C02439=-605,59585,-14,-1321,-34531,-989
C02440=-605,59585,1386,-1321,-34531,-989
C02441=-133,59559,1353,-1384,-34516,-1179
C02442=-133,59559,-47,-1384,-34516,-1179
C02443=-94,59556,-50,-1389,-34515,-1194
C02444=-94,59556,1350,-1389,-34515,-1194
C02445=167,59542,1332,-1423,-34507,-1299
C02446=167,59542,-68,-1423,-34507,-1299
C02447=216,59539,-71,-1430,-34505,-1318
C02448=216,59539,1329,-1430,-34505,-1318
C02449=494,59523,1310,-1467,-34497,-1430
C02450=494,59523,-90,-1467,-34497,-1430
C02451=533,59521,-93,-1472,-34495,-1445
C02452=533,59521,1307,-1472,-34495,-1445
C02453=638,59515,1300,-1486,-34492,-1488
C02454=638,59515,-100,-1486,-34492,-1488
C02455=681,59512,-103,-1492,-34491,-1505
C02456=681,59512,1297,-1492,-34491,-1505
C02457=1167,59485,1263,-1556,-34476,-1699
C02458=1167,59485,-137,-1556,-34476,-1699
C02459=1205,59483,-140,-1561,-34474,-1715
C02460=1205,59483,1260,-1561,-34474,-1715
C02461=-5420,59813,1651,-682,-34655,941
C02462=-5420,59813,251,-682,-34655,941
C02463=-5370,59811,248,-689,-34654,922
C02464=-5370,59811,1648,-689,-34654,922
C02465=-4567,59765,1592,-795,-34629,600
C02466=-4567,59765,192,-795,-34629,600
C02467=-4511,59762,188,-803,-34627,577
C02468=-4511,59762,1588,-803,-34627,577
C02469=-4166,59743,1565,-849,-34616,439
C02470=-4166,59743,165,-849,-34616,439
C02471=-4106,59739,160,-857,-34614,415
C02472=-4106,59739,1560,-857,-34614,415
C02473=-3314,59694,1506,-962,-34589,97
C02474=-3314,59694,106,-962,-34589,97
C02475=-3268,59692,102,-968,-34588,79
C02476=-3268,59692,1502,-968,-34588,79
C02477=-2546,59651,1453,-1064,-34565,-211
C02478=-2546,59651,53,-1064,-34565,-211
C02479=-2500,59648,49,-1070,-34564,-229
C02480=-2500,59648,1449,-1070,-34564,-229
C02481=-2225,59633,1430,-1106,-34555,-339
C02482=-2225,59633,30,-1106,-34555,-339
C02483=-2173,59630,27,-1114,-34553,-360
C02484=-2173,59630,1427,-1114,-34553,-360
C02485=-1937,59617,1411,-1145,-34546,-455
C02486=-1937,59617,11,-1145,-34546,-455
C02487=-1891,59614,7,-1151,-34544,-473
C02488=-1891,59614,1407,-1151,-34544,-473
C02489=-1729,59605,1396,-1172,-34539,-538
C02490=-1729,59605,-4,-1172,-34539,-538
C02491=-1687,59602,-7,-1178,-34538,-555
C02492=-1687,59602,1393,-1178,-34538,-555
C02493=-1606,59598,1388,-1189,-34535,-588
C02494=-1606,59598,-12,-1189,-34535,-588
C02495=-1556,59595,-16,-1195,-34534,-607
C02496=-1556,59595,1384,-1195,-34534,-607
C02497=-1412,59587,1374,-1215,-34529,-665
C02498=-1412,59587,-26,-1215,-34529,-665
C02499=-1331,59582,-31,-1225,-34527,-698
C02500=-1331,59582,1369,-1225,-34527,-698
C02501=-1250,59578,1363,-1236,-34524,-730
C02502=-1250,59578,-37,-1236,-34524,-730
C02503=-1165,59573,-43,-1247,-34522,-764
C02504=-1165,59573,1357,-1247,-34522,-764
C02505=-1056,59567,1350,-1262,-34518,-808
C02506=-1056,59567,-50,-1262,-34518,-808
C02507=-1010,59564,-53,-1268,-34517,-826
C02508=-1010,59564,1347,-1268,-34517,-826
C02509=-655,59544,1322,-1315,-34506,-969
C02510=-655,59544,-78,-1315,-34506,-969
C02511=-619,59542,-80,-1320,-34504,-983
C02512=-619,59542,1320,-1320,-34504,-983
C02513=-130,59514,1286,-1385,-34489,-1179
C02514=-130,59514,-114,-1385,-34489,-1179
C02515=-95,59512,-117,-1390,-34488,-1193
C02516=-95,59512,1283,-1390,-34488,-1193
C02517=173,59497,1265,-1425,-34480,-1301
C02518=173,59497,-135,-1425,-34480,-1301
C02519=219,59495,-138,-1431,-34478,-1319
C02520=219,59495,1262,-1431,-34478,-1319
C02521=497,59479,1242,-1468,-34469,-1430
C02522=497,59479,-158,-1468,-34469,-1430
C02523=539,59477,-161,-1474,-34468,-1447
C02524=539,59477,1239,-1474,-34468,-1447
C02525=648,59470,1232,-1488,-34465,-1491
C02526=648,59470,-168,-1488,-34465,-1491
C02527=691,59468,-171,-1494,-34463,-1508
C02528=691,59468,1229,-1494,-34463,-1508
C02529=1170,59441,1196,-1557,-34448,-1700
C02530=1170,59441,-204,-1557,-34448,-1700
C02531=1208,59439,-207,-1563,-34447,-1716
C02532=1208,59439,1193,-1563,-34447,-1716
C02533=-5403,59768,1583,-685,-34628,935
C02534=-5403,59768,183,-685,-34628,935
C02535=-5354,59765,179,-692,-34626,915
C02536=-5354,59765,1579,-692,-34626,915
C02537=-4551,59720,1524,-798,-34601,594
C02538=-4551,59720,124,-798,-34601,594
C02539=-4494,59717,120,-806,-34599,571
C02540=-4494,59717,1520,-806,-34599,571
C02541=-4195,59700,1499,-846,-34590,451
C02542=-4195,59700,99,-846,-34590,451
C02543=-4128,59696,95,-854,-34588,424
C02544=-4128,59696,1495,-854,-34588,424
C02545=-3332,59651,1440,-960,-34563,105
C02546=-3332,59651,40,-960,-34563,105
C02547=-3283,59648,36,-967,-34561,85
C02548=-3283,59648,1436,-967,-34561,85
C02549=-2543,59607,1385,-1065,-34538,-211
C02550=-2543,59607,-15,-1065,-34538,-211
C02551=-2494,59604,-18,-1072,-34536,-231
C02552=-2494,59604,1382,-1072,-34536,-231
C02553=-2226,59589,1363,-1107,-34528,-338
C02554=-2226,59589,-37,-1107,-34528,-338
C02555=-2177,59586,-40,-1114,-34526,-358
C02556=-2177,59586,1360,-1114,-34526,-358
C02557=-1920,59571,1342,-1148,-34518,-461
C02558=-1920,59571,-58,-1148,-34518,-461
C02559=-1870,59569,-61,-1154,-34517,-481
C02560=-1870,59569,1339,-1154,-34517,-481
C02561=-1758,59562,1331,-1169,-34513,-526
C02562=-1758,59562,-69,-1169,-34513,-526
C02563=-1715,59560,-72,-1175,-34512,-543
C02564=-1715,59560,1328,-1175,-34512,-543
C02565=-1599,59553,1320,-1190,-34508,-590
C02566=-1599,59553,-80,-1190,-34508,-590
C02567=-1532,59549,-84,-1199,-34506,-616
C02568=-1532,59549,1316,-1199,-34506,-616
C02569=-1370,59540,1304,-1221,-34501,-681
C02570=-1370,59540,-96,-1221,-34501,-681
C02571=-1226,59532,-106,-1240,-34496,-739
C02572=-1226,59532,1294,-1240,-34496,-739
C02573=-1039,59522,1282,-1265,-34491,-814
C02574=-1039,59522,-118,-1265,-34491,-814
C02575=-986,59519,-122,-1272,-34489,-835
C02576=-986,59519,1278,-1272,-34489,-835
C02577=-684,59502,1257,-1312,-34479,-957
C02578=-684,59502,-143,-1312,-34479,-957
C02579=-641,59499,-146,-1318,-34478,-973
C02580=-641,59499,1254,-1318,-34478,-973
C02581=-131,59470,1219,-1386,-34462,-1178
C02582=-131,59470,-181,-1386,-34462,-1178
C02583=-92,59468,-184,-1391,-34461,-1194
C02584=-92,59468,1216,-1391,-34461,-1194
C02585=176,59453,1198,-1426,-34452,-1301
C02586=176,59453,-202,-1426,-34452,-1301
C02587=222,59450,-206,-1432,-34451,-1319
C02588=222,59450,1194,-1432,-34451,-1319
C02589=503,59435,1175,-1470,-34442,-1432
C02590=503,59435,-225,-1470,-34442,-1432
C02591=542,59432,-228,-1475,-34441,-1448
C02592=542,59432,1172,-1475,-34441,-1448
C02593=655,59426,1165,-1490,-34437,-1493
C02594=655,59426,-235,-1490,-34437,-1493
C02595=697,59424,-238,-1496,-34436,-1510
C02596=697,59424,1162,-1496,-34436,-1510
C02597=827,59416,1153,-1513,-34432,-1562
C02598=827,59416,-247,-1513,-34432,-1562
C02599=848,59415,-249,-1516,-34431,-1571
C02600=848,59415,1151,-1516,-34431,-1571
C02601=1165,59397,1129,-1558,-34421,-1698
C02602=1165,59397,-271,-1558,-34421,-1698
C02603=1204,59395,-273,-1563,-34420,-1713
C02604=1204,59395,1127,-1563,-34420,-1713
C02605=-5393,59723,1515,-687,-34601,932
C02606=-5393,59723,115,-687,-34601,932
C02607=-5341,59720,111,-694,-34599,911
C02608=-5341,59720,1511,-694,-34599,911
C02609=-4534,59675,1456,-801,-34574,587
C02610=-4534,59675,56,-801,-34574,587
C02611=-4474,59671,52,-809,-34572,563
C02612=-4474,59671,1452,-809,-34572,563
C02613=-4221,59657,1434,-843,-34564,462
C02614=-4221,59657,34,-843,-34564,462
C02615=-4157,59653,30,-851,-34562,436
C02616=-4157,59653,1430,-851,-34562,436
C02617=-3344,59607,1374,-959,-34536,110
C02618=-3344,59607,-26,-959,-34536,110
C02619=-3298,59605,-30,-965,-34535,92
C02620=-3298,59605,1370,-965,-34535,92
C02621=-2544,59562,1318,-1066,-34511,-210
C02622=-2544,59562,-82,-1066,-34511,-210
C02623=-2498,59560,-85,-1072,-34509,-229
C02624=-2498,59560,1315,-1072,-34509,-229
C02625=-2227,59544,1296,-1108,-34501,-337
C02626=-2227,59544,-104,-1108,-34501,-337
C02627=-2178,59542,-107,-1114,-34499,-357
C02628=-2178,59542,1293,-1114,-34499,-357
C02629=-1892,59526,1273,-1152,-34490,-471
C02630=-1892,59526,-127,-1152,-34490,-471
C02631=-1741,59517,-137,-1172,-34486,-532
C02632=-1741,59517,1263,-1172,-34486,-532
C02633=-1019,59476,1213,-1268,-34463,-822
C02634=-1019,59476,-187,-1268,-34463,-822
C02635=-941,59472,-192,-1279,-34460,-853
C02636=-941,59472,1208,-1279,-34460,-853
C02637=-723,59460,1193,-1308,-34453,-940
C02638=-723,59460,-207,-1308,-34453,-940
C02639=-667,59457,-211,-1315,-34452,-963
C02640=-667,59457,1189,-1315,-34452,-963
C02641=-135,59427,1152,-1386,-34435,-1176
C02642=-135,59427,-248,-1386,-34435,-1176
C02643=-89,59424,-251,-1392,-34433,-1194
C02644=-89,59424,1149,-1392,-34433,-1194
C02645=175,59409,1131,-1427,-34425,-1300
C02646=175,59409,-269,-1427,-34425,-1300
C02647=221,59406,-273,-1433,-34424,-1318
C02648=221,59406,1127,-1433,-34424,-1318
C02649=506,59390,1108,-1471,-34415,-1433
C02650=506,59390,-292,-1471,-34415,-1433
C02651=541,59388,-295,-1476,-34414,-1447
C02652=541,59388,1105,-1476,-34414,-1447
C02653=661,59382,1097,-1492,-34410,-1495
C02654=661,59382,-303,-1492,-34410,-1495
C02655=707,59379,-306,-1498,-34408,-1513
C02656=707,59379,1094,-1498,-34408,-1513
C02657=830,59372,1085,-1514,-34404,-1563
C02658=830,59372,-315,-1514,-34404,-1563
C02659=855,59371,-316,-1517,-34404,-1573
C02660=855,59371,1084,-1517,-34404,-1573
C02661=1154,59354,1063,-1557,-34394,-1693
C02662=1154,59354,-337,-1557,-34394,-1693
C02663=1197,59351,-340,-1563,-34393,-1710
C02664=1197,59351,1060,-1563,-34393,-1710
C02665=-5380,59678,1447,-689,-34573,927
C02666=-5380,59678,47,-689,-34573,927
C02667=-5320,59674,43,-697,-34571,903
C02668=-5320,59674,1443,-697,-34571,903
C02669=-4517,59629,1388,-804,-34546,581
C02670=-4517,59629,-12,-804,-34546,581
C02671=-4443,59625,-18,-814,-34544,552
C02672=-4443,59625,1382,-814,-34544,552
C02673=-4257,59614,1370,-839,-34538,477
C02674=-4257,59614,-30,-839,-34538,477
C02675=-4183,59610,-36,-849,-34536,447
C02676=-4183,59610,1364,-849,-34536,447
C02677=-3362,59564,1308,-958,-34510,118
C02678=-3362,59564,-92,-958,-34510,118
C02679=-3316,59562,-95,-964,-34508,100
C02680=-3316,59562,1305,-964,-34508,100
C02681=-2221,59500,1229,-1109,-34474,-339
C02682=-2221,59500,-171,-1109,-34474,-339
C02683=-2193,59498,-173,-1113,-34473,-351
C02684=-2193,59498,1227,-1113,-34473,-351
C02685=-991,59431,1144,-1273,-34435,-832
C02686=-991,59431,-256,-1273,-34435,-832
C02687=-699,59414,-276,-1312,-34426,-949
C02688=-699,59414,1124,-1312,-34426,-949
C02689=-136,59383,1085,-1386,-34408,-1175
C02690=-136,59383,-315,-1386,-34408,-1175
C02691=-86,59380,-318,-1393,-34406,-1195
C02692=-86,59380,1082,-1393,-34406,-1195
C02693=178,59365,1063,-1428,-34398,-1301
C02694=178,59365,-337,-1428,-34398,-1301
C02695=224,59362,-340,-1434,-34396,-1319
C02696=224,59362,1060,-1434,-34396,-1319
C02697=509,59346,1041,-1472,-34387,-1433
C02698=509,59346,-359,-1472,-34387,-1433
C02699=544,59344,-362,-1477,-34386,-1447
C02700=544,59344,1038,-1477,-34386,-1447
C02701=664,59337,1030,-1493,-34383,-1495
C02702=664,59337,-370,-1493,-34383,-1495
C02703=710,59335,-373,-1499,-34381,-1514
C02704=710,59335,1027,-1499,-34381,-1514
C02705=837,59328,1018,-1516,-34377,-1565
C02706=837,59328,-382,-1516,-34377,-1565
C02707=868,59326,-384,-1520,-34376,-1577
C02708=868,59326,1016,-1520,-34376,-1577
C02709=1136,59311,997,-1555,-34368,-1685
C02710=1136,59311,-403,-1555,-34368,-1685
C02711=1185,59308,-406,-1562,-34366,-1704
C02712=1185,59308,994,-1562,-34366,-1704
C02713=-5360,59632,1379,-693,-34546,920
C02714=-5360,59632,-21,-693,-34546,920
C02715=-5304,59629,-25,-700,-34544,897
C02716=-5304,59629,1375,-700,-34544,897
C02717=-4490,59583,1319,-808,-34518,571
C02718=-4490,59583,-81,-808,-34518,571
C02719=-4384,59577,-89,-822,-34515,529
C02720=-4384,59577,1311,-822,-34515,529
C02721=-4325,59574,1307,-830,-34513,505
C02722=-4325,59574,-93,-830,-34513,505
C02723=-4219,59568,-100,-844,-34510,462
C02724=-4219,59568,1300,-844,-34510,462
C02725=-3381,59521,1242,-956,-34483,126
C02726=-3381,59521,-158,-956,-34483,126
C02727=-3331,59518,-161,-962,-34482,106
C02728=-3331,59518,1239,-962,-34482,106
C02729=-901,59381,1071,-1285,-34405,-868
C02730=-901,59381,-329,-1285,-34405,-868
C02731=-784,59375,-337,-1301,-34401,-914
C02732=-784,59375,1063,-1301,-34401,-914
C02733=-126,59338,1017,-1389,-34380,-1178
C02734=-126,59338,-383,-1389,-34380,-1178
C02735=-94,59336,-385,-1393,-34379,-1191
C02736=-94,59336,1015,-1393,-34379,-1191
C02737=181,59321,996,-1429,-34371,-1301
C02738=181,59321,-404,-1429,-34371,-1301
C02739=227,59318,-407,-1435,-34369,-1320
C02740=227,59318,993,-1435,-34369,-1320
C02741=508,59302,974,-1473,-34360,-1432
C02742=508,59302,-426,-1473,-34360,-1432
C02743=561,59299,-430,-1480,-34359,-1454
C02744=561,59299,970,-1480,-34359,-1454
C02745=843,59283,951,-1517,-34350,-1567
C02746=843,59283,-449,-1517,-34350,-1567
C02747=878,59281,-452,-1522,-34349,-1581
C02748=878,59281,948,-1522,-34349,-1581
C02749=1107,59269,932,-1552,-34341,-1672
C02750=1107,59269,-468,-1552,-34341,-1672
C02751=1164,59265,-472,-1560,-34340,-1695
C02752=1164,59265,928,-1560,-34340,-1695
C02753=-5340,59586,1310,-696,-34518,912
C02754=-5340,59586,-90,-696,-34518,912
C02755=-5277,59583,-94,-704,-34516,887
C02756=-5277,59583,1306,-704,-34516,887
C02757=-4452,59537,1249,-814,-34490,556
C02758=-4452,59537,-151,-814,-34490,556
C02759=-4269,59526,-164,-838,-34484,483
C02760=-4269,59526,1236,-838,-34484,483
C02761=-3403,59478,1176,-954,-34457,136
C02762=-3403,59478,-224,-954,-34457,136
C02763=-3353,59475,-227,-960,-34455,116
C02764=-3353,59475,1173,-960,-34455,116
C02765=511,59258,906,-1474,-34333,-1433
C02766=511,59258,-494,-1474,-34333,-1433
C02767=561,59255,-497,-1481,-34331,-1453
C02768=561,59255,903,-1481,-34331,-1453
C02769=853,59239,883,-1519,-34322,-1570
C02770=853,59239,-517,-1519,-34322,-1570
C02771=902,59236,-521,-1526,-34321,-1590
C02772=902,59236,879,-1526,-34321,-1590
C02773=1057,59227,869,-1547,-34316,-1652
C02774=1057,59227,-531,-1547,-34316,-1652
C02775=1138,59223,-537,-1557,-34313,-1684
C02776=1138,59223,863,-1557,-34313,-1684
C02777=-5313,59540,1241,-700,-34490,902
C02778=-5313,59540,-159,-700,-34490,902
C02779=-5253,59537,-163,-708,-34489,878
C02780=-5253,59537,1237,-708,-34489,878
C02781=-3418,59434,1110,-952,-34430,142
C02782=-3418,59434,-290,-952,-34430,142
C02783=-3375,59432,-292,-958,-34429,125
C02784=-3375,59432,1108,-958,-34429,125
C02785=874,59194,814,-1523,-34294,-1578
C02786=874,59194,-586,-1523,-34294,-1578
C02787=1103,59181,-601,-1553,-34287,-1669
C02788=1103,59181,799,-1553,-34287,-1669
C02789=1508,59158,771,-1607,-34274,-1832
C02790=1508,59158,-629,-1607,-34274,-1832
C02791=1532,59157,-631,-1611,-34273,-1842
C02792=1532,59157,769,-1611,-34273,-1842
C02793=-5293,59495,1173,-704,-34463,894
C02794=-5293,59495,-227,-704,-34463,894
C02795=-5229,59491,-232,-712,-34461,869
C02796=-5229,59491,1168,-712,-34461,869
C02797=-3440,59391,1045,-950,-34404,151
C02798=-3440,59391,-355,-950,-34404,151
C02799=-3387,59388,-359,-957,-34402,130
C02800=-3387,59388,1041,-957,-34402,130
C02801=915,59148,745,-1529,-34266,-1594
C02802=915,59148,-655,-1529,-34266,-1594
C02803=1038,59141,-664,-1546,-34262,-1643
C02804=1038,59141,736,-1546,-34262,-1643
C02805=1482,59116,705,-1605,-34248,-1821
C02806=1482,59116,-695,-1605,-34248,-1821
C02807=1567,59111,-700,-1616,-34245,-1855
C02808=1567,59111,700,-1616,-34245,-1855
C02809=-5266,59449,1104,-708,-34435,884
C02810=-5266,59449,-296,-708,-34435,884
C02811=-5202,59445,-301,-716,-34433,858
C02812=-5202,59445,1099,-716,-34433,858
C02813=-3458,59348,979,-948,-34378,159
C02814=-3458,59348,-421,-948,-34378,159
C02815=-3405,59345,-424,-955,-34376,138
C02816=-3405,59345,976,-955,-34376,138
C02817=1485,59072,638,-1606,-34221,-1821
C02818=1485,59072,-762,-1606,-34221,-1821
C02819=1538,59069,-765,-1613,-34219,-1843
C02820=1538,59069,635,-1613,-34219,-1843
C02821=-5245,59403,1035,-711,-34408,876
C02822=-5245,59403,-365,-711,-34408,876
C02823=-5178,59399,-369,-720,-34405,849
C02824=-5178,59399,1031,-720,-34405,849
C02825=-3484,59305,914,-946,-34351,170
C02826=-3484,59305,-486,-946,-34351,170
C02827=-3424,59302,-490,-954,-34350,146
C02828=-3424,59302,910,-954,-34350,146
C02829=-5215,59357,966,-716,-34380,864
C02830=-5215,59357,-434,-716,-34380,864
C02831=-5155,59354,-438,-724,-34378,840
C02832=-5155,59354,962,-724,-34378,840
C02833=-3516,59262,849,-942,-34325,184
C02834=-3516,59262,-551,-942,-34325,184
C02835=-3460,59259,-555,-949,-34324,161
C02836=-3460,59259,845,-949,-34324,161
C02837=-5184,59311,897,-721,-34352,853
C02838=-5184,59311,-503,-721,-34352,853
C02839=-5117,59307,-508,-730,-34350,826
C02840=-5117,59307,892,-730,-34350,826
C02841=-3552,59220,784,-938,-34300,199
C02842=-3552,59220,-616,-938,-34300,199
C02843=-3482,59216,-620,-947,-34297,171
C02844=-3482,59216,780,-947,-34297,171
C02845=-5157,59265,828,-725,-34324,842
C02846=-5157,59265,-572,-725,-34324,842
C02847=-5076,59260,-578,-736,-34321,810
C02848=-5076,59260,822,-736,-34321,810
C02849=-3592,59178,720,-933,-34274,215
C02850=-3592,59178,-680,-933,-34274,215
C02851=-3518,59174,-685,-943,-34272,186
C02852=-3518,59174,715,-943,-34272,186
C02853=-5119,59218,758,-731,-34296,828
C02854=-5119,59218,-642,-731,-34296,828
C02855=-5041,59214,-647,-741,-34293,797
C02856=-5041,59214,753,-741,-34293,797
C02857=-3635,59136,656,-928,-34248,233
C02858=-3635,59136,-744,-928,-34248,233
C02859=-3558,59132,-749,-939,-34246,202
C02860=-3558,59132,651,-939,-34246,202
C02861=-5081,59172,689,-736,-34268,813
C02862=-5081,59172,-711,-736,-34268,813
C02863=-4965,59165,-719,-752,-34264,766
C02864=-4965,59165,681,-752,-34264,766
C02865=-3678,59094,592,-923,-34223,251
C02866=-3678,59094,-808,-923,-34223,251
C02867=-3597,59090,-814,-934,-34220,219
C02868=-3597,59090,586,-934,-34220,219
C02869=-5036,59125,618,-743,-34239,796
C02870=-5036,59125,-782,-743,-34239,796
C02871=-4888,59117,-792,-763,-34234,736
C02872=-4888,59117,608,-763,-34234,736
C02873=-3736,59053,529,-916,-34197,275
C02874=-3736,59053,-871,-916,-34197,275
C02875=-3648,59048,-877,-928,-34195,239
C02876=-3648,59048,523,-928,-34195,239
C02877=-4953,59076,546,-755,-34210,763
C02878=-4953,59076,-854,-755,-34210,763
C02879=-4819,59068,-864,-773,-34205,709
C02880=-4819,59068,536,-773,-34205,709
C02881=-3782,59011,465,-911,-34172,294
C02882=-3782,59011,-935,-911,-34172,294
C02883=-3694,59006,-941,-922,-34169,259
C02884=-3694,59006,459,-922,-34169,259
C02885=-4880,59027,473,-765,-34180,734
C02886=-4880,59027,-927,-765,-34180,734
C02887=-4739,59019,-936,-784,-34176,677
C02888=-4739,59019,464,-784,-34176,677
C02889=-3840,58970,402,-904,-34147,317
C02890=-3840,58970,-998,-904,-34147,317
C02891=-3748,58965,-1004,-916,-34144,281
C02892=-3748,58965,396,-916,-34144,281
C02893=-4800,58978,401,-777,-34151,702
C02894=-4800,58978,-999,-777,-34151,702
C02895=-4609,58968,-1012,-802,-34145,626
C02896=-4609,58968,388,-802,-34145,626
C02897=-3925,58930,341,-893,-34123,352
C02898=-3925,58930,-1059,-893,-34123,352
C02899=-3802,58923,-1068,-910,-34119,303
C02900=-3802,58923,332,-910,-34119,303
C02901=-4695,58928,327,-791,-34120,661
C02902=-4695,58928,-1073,-791,-34120,661
C02903=-4462,58915,-1089,-822,-34113,568
C02904=-4462,58915,311,-822,-34113,568
C02905=-4194,58901,292,-858,-34104,460
C02906=-4194,58901,-1108,-858,-34104,460
C02907=-3873,58883,-1130,-901,-34094,332
C02908=-3873,58883,270,-901,-34094,332
C02909=-4537,58875,249,-813,-34088,598
C02910=-4537,58875,-1151,-813,-34088,598
C02911=-3991,58845,-1189,-886,-34071,379
C02912=-3991,58845,211,-886,-34071,379
C02913=-4485,58828,178,-821,-34060,578
C02914=-4485,58828,-1222,-821,-34060,578
C02915=-4330,58819,-1233,-841,-34055,516
C02916=-4330,58819,167,-841,-34055,516
C02917=-4493,58784,112,-820,-34033,582
C02918=-4493,58784,-1288,-820,-34033,582
C02919=-4430,58780,-1293,-829,-34031,556
C02920=-4430,58780,107,-829,-34031,556
C02921=-4494,58739,44,-821,-34006,583
C02922=-4494,58739,-1356,-821,-34006,583
C02923=-4427,58736,-1360,-830,-34004,556
C02924=-4427,58736,40,-830,-34004,556
C02925=-4492,58695,-23,-822,-33979,582
C02926=-4492,58695,-1423,-822,-33979,582
C02927=-4428,58691,-1427,-830,-33977,557
C02928=-4428,58691,-27,-830,-33977,557
C02929=-4478,58650,-91,-824,-33952,577
C02930=-4478,58650,-1491,-824,-33952,577
C02931=-4422,58647,-1495,-832,-33950,555
C02932=-4422,58647,-95,-832,-33950,555
C02933=-4472,58605,-158,-826,-33924,576
C02934=-4472,58605,-1558,-826,-33924,576
C02935=-4388,58600,-1564,-837,-33922,542
C02936=-4388,58600,-164,-837,-33922,542
C02937=-4473,58560,-225,-826,-33898,576
C02938=-4473,58560,-1625,-826,-33898,576
C02939=-4371,58555,-1632,-840,-33894,535
C02940=-4371,58555,-232,-840,-33894,535
C02941=-4485,58517,-292,-825,-33871,582
C02942=-4485,58517,-1692,-825,-33871,582
C02943=-4344,58509,-1701,-844,-33866,525
C02944=-4344,58509,-301,-844,-33866,525
C02945=-4503,58473,-357,-824,-33845,590
C02946=-4503,58473,-1757,-824,-33845,590
C02947=-4419,58469,-1763,-835,-33842,556
C02948=-4419,58469,-363,-835,-33842,556
C02949=-4387,58467,-365,-839,-33841,543
C02950=-4387,58467,-1765,-839,-33841,543
C02951=-4309,58463,-1771,-849,-33838,512
C02952=-4309,58463,-371,-849,-33838,512
C02953=-4526,58430,-423,-821,-33818,599
C02954=-4526,58430,-1823,-821,-33818,599
C02955=-4416,58424,-1830,-836,-33815,555
C02956=-4416,58424,-430,-836,-33815,555
C02957=-4349,58421,-435,-845,-33813,528
C02958=-4349,58421,-1835,-845,-33813,528
C02959=-4279,58417,-1840,-854,-33810,500
C02960=-4279,58417,-440,-854,-33810,500
C02961=-4548,58387,-488,-819,-33792,608
C02962=-4548,58387,-1888,-819,-33792,608
C02963=-4491,58384,-1892,-827,-33790,586
C02964=-4491,58384,-492,-827,-33790,586
C02965=-4463,58382,-494,-830,-33789,574
C02966=-4463,58382,-1894,-830,-33789,574
C02967=-4417,58380,-1897,-836,-33788,556
C02968=-4417,58380,-497,-836,-33788,556
C02969=-4315,58374,-504,-850,-33785,515
C02970=-4315,58374,-1904,-850,-33785,515
C02971=-4244,58370,-1909,-859,-33782,487
C02972=-4244,58370,-509,-859,-33782,487
C02973=-4570,58344,-554,-817,-33766,618
C02974=-4570,58344,-1954,-817,-33766,618
C02975=-4510,58340,-1958,-825,-33764,594
C02976=-4510,58340,-558,-825,-33764,594
C02977=-4464,58338,-561,-831,-33762,575
C02978=-4464,58338,-1961,-831,-33762,575
C02979=-4418,58335,-1964,-837,-33761,557
C02980=-4418,58335,-564,-837,-33761,557
C02981=-4284,58328,-574,-855,-33757,503
C02982=-4284,58328,-1974,-855,-33757,503
C02983=-4213,58324,-1978,-864,-33754,475
C02984=-4213,58324,-578,-864,-33754,475
C02985=-4599,58301,-619,-813,-33740,630
C02986=-4599,58301,-2019,-813,-33740,630
C02987=-4546,58298,-2023,-821,-33738,609
C02988=-4546,58298,-623,-821,-33738,609
C02989=-4461,58293,-628,-832,-33735,575
C02990=-4461,58293,-2028,-832,-33735,575
C02991=-4415,58291,-2032,-838,-33734,557
C02992=-4415,58291,-632,-838,-33734,557
C02993=-4250,58282,-643,-860,-33728,490
C02994=-4250,58282,-2043,-860,-33728,490
C02995=-4186,58279,-2047,-869,-33726,465
C02996=-4186,58279,-647,-869,-33726,465
C02997=-4621,58257,-685,-811,-33714,639
C02998=-4621,58257,-2085,-811,-33714,639
C02999=-4575,58255,-2088,-817,-33712,621
C03000=-4575,58255,-688,-817,-33712,621
C03001=-4459,58249,-696,-833,-33708,574
C03002=-4459,58249,-2096,-833,-33708,574
C03003=-4416,58246,-2099,-839,-33707,557
C03004=-4416,58246,-699,-839,-33707,557
C03005=-4222,58236,-712,-864,-33701,480
C03006=-4222,58236,-2112,-864,-33701,480
C03007=-4152,58232,-2117,-874,-33698,452
C03008=-4152,58232,-717,-874,-33698,452
C03009=-4650,58215,-750,-808,-33688,652
C03010=-4650,58215,-2150,-808,-33688,652
C03011=-4597,58212,-2153,-815,-33686,630
C03012=-4597,58212,-753,-815,-33686,630
C03013=-4460,58204,-763,-833,-33681,575
C03014=-4460,58204,-2163,-833,-33681,575
C03015=-4421,58202,-2165,-839,-33680,560
C03016=-4421,58202,-765,-839,-33680,560
C03017=-4188,58190,-781,-870,-33672,467
C03018=-4188,58190,-2181,-870,-33672,467
C03019=-4107,58185,-2187,-881,-33670,434
C03020=-4107,58185,-787,-881,-33670,434
C03021=-4683,58172,-815,-804,-33662,665
C03022=-4683,58172,-2215,-804,-33662,665
C03023=-4627,58169,-2218,-812,-33660,643
C03024=-4627,58169,-818,-812,-33660,643
C03025=-4461,58160,-830,-834,-33654,576
C03026=-4461,58160,-2230,-834,-33654,576
C03027=-4418,58158,-2233,-840,-33653,559
C03028=-4418,58158,-833,-840,-33653,559
C03029=-4150,58143,-851,-875,-33644,452
C03030=-4150,58143,-2251,-875,-33644,452
C03031=-4069,58139,-2257,-886,-33642,419
C03032=-4069,58139,-857,-886,-33642,419
C03033=-4716,58129,-879,-801,-33636,679
C03034=-4716,58129,-2279,-801,-33636,679
C03035=-4659,58126,-2283,-808,-33634,656
C03036=-4659,58126,-883,-808,-33634,656
C03037=-4458,58115,-897,-835,-33627,576
C03038=-4458,58115,-2297,-835,-33627,576
C03039=-4419,58113,-2300,-840,-33626,560
C03040=-4419,58113,-900,-840,-33626,560
C03041=-4102,58096,-921,-883,-33616,433
C03042=-4102,58096,-2321,-883,-33616,433
C03043=-4035,58093,-2326,-892,-33613,406
C03044=-4035,58093,-926,-892,-33613,406
C03045=-4745,58086,-944,-797,-33610,691
C03046=-4745,58086,-2344,-797,-33610,691
C03047=-4692,58084,-2348,-804,-33608,670
C03048=-4692,58084,-948,-804,-33608,670
C03049=-4459,58071,-964,-836,-33600,577
C03050=-4459,58071,-2364,-836,-33600,577
C03051=-4417,58069,-2367,-841,-33599,560
C03052=-4417,58069,-967,-841,-33599,560
C03053=-4064,58050,-991,-888,-33587,418
C03054=-4064,58050,-2391,-888,-33587,418
C03055=-3990,58046,-2396,-898,-33585,389
C03056=-3990,58046,-996,-898,-33585,389
C03057=-4785,58044,-1009,-793,-33584,708
C03058=-4785,58044,-2409,-793,-33584,708
C03059=-4725,58041,-2413,-801,-33582,683
C03060=-4725,58041,-1013,-801,-33582,683
C03061=-4456,58027,-1031,-837,-33573,576
C03062=-4456,58027,-2431,-837,-33573,576
C03063=-4414,58024,-2434,-842,-33572,559
C03064=-4414,58024,-1034,-842,-33572,559
C03065=-4019,58003,-1061,-895,-33559,401
C03066=-4019,58003,-2461,-895,-33559,401
C03067=-3938,57999,-2467,-906,-33556,369
C03068=-3938,57999,-1067,-906,-33556,369
C03069=-4817,58001,-1074,-789,-33558,721
C03070=-4817,58001,-2474,-789,-33558,721
C03071=-4765,57998,-2477,-796,-33557,700
C03072=-4765,57998,-1077,-796,-33557,700
C03073=-4454,57982,-1099,-838,-33546,576
C03074=-4454,57982,-2499,-838,-33546,576
C03075=-4411,57980,-2501,-843,-33545,559
C03076=-4411,57980,-1101,-843,-33545,559
C03077=-3977,57957,-1131,-901,-33531,385
C03078=-3977,57957,-2531,-901,-33531,385
C03079=-3900,57953,-2536,-912,-33528,354
C03080=-3900,57953,-1136,-912,-33528,354
C03081=-4850,57959,-1138,-785,-33533,735
C03082=-4850,57959,-2538,-785,-33533,735
C03083=-4797,57956,-2542,-792,-33531,714
C03084=-4797,57956,-1142,-792,-33531,714
C03085=-4455,57938,-1166,-838,-33519,577
C03086=-4455,57938,-2566,-838,-33519,577
C03087=-4412,57935,-2568,-844,-33518,560
C03088=-4412,57935,-1168,-844,-33518,560
C03089=-3936,57910,-1201,-908,-33502,369
C03090=-3936,57910,-2601,-908,-33502,369
C03091=-3858,57906,-2606,-918,-33500,338
C03092=-3858,57906,-1206,-918,-33500,338
C03093=-4887,57916,-1203,-781,-33507,750
C03094=-4887,57916,-2603,-781,-33507,750
C03095=-4837,57913,-2606,-788,-33505,730
C03096=-4837,57913,-1206,-788,-33505,730
C03097=-4452,57893,-1233,-839,-33492,576
C03098=-4452,57893,-2633,-839,-33492,576
C03099=-4413,57891,-2635,-844,-33491,561
C03100=-4413,57891,-1235,-844,-33491,561
C03101=-3894,57864,-1271,-914,-33474,353
C03102=-3894,57864,-2671,-914,-33474,353
C03103=-3817,57859,-2676,-924,-33471,322
C03104=-3817,57859,-1276,-924,-33471,322
C03105=-4923,57874,-1268,-777,-33481,765
C03106=-4923,57874,-2668,-777,-33481,765
C03107=-4870,57871,-2671,-784,-33479,744
C03108=-4870,57871,-1271,-784,-33479,744
C03109=-4453,57849,-1300,-840,-33465,577
C03110=-4453,57849,-2700,-840,-33465,577
C03111=-4414,57847,-2702,-845,-33464,561
C03112=-4414,57847,-1302,-845,-33464,561
C03113=-3856,57817,-1341,-920,-33446,338
C03114=-3856,57817,-2741,-920,-33446,338
C03115=-3765,57812,-2747,-932,-33443,302
C03116=-3765,57812,-1347,-932,-33443,302
C03117=-4963,57831,-1332,-772,-33455,781
C03118=-4963,57831,-2732,-772,-33455,781
C03119=-4906,57828,-2736,-780,-33454,759
C03120=-4906,57828,-1336,-780,-33454,759
C03121=-4451,57804,-1367,-841,-33438,576
C03122=-4451,57804,-2767,-841,-33438,576
C03123=-4412,57802,-2770,-846,-33437,561
C03124=-4412,57802,-1370,-846,-33437,561
C03125=-3819,57771,-1410,-925,-33417,324
C03126=-3819,57771,-2810,-925,-33417,324
C03127=-3730,57766,-2816,-937,-33414,288
C03128=-3730,57766,-1416,-937,-33414,288
C03129=-5006,57789,-1396,-767,-33430,799
C03130=-5006,57789,-2796,-767,-33430,799
C03131=-4946,57786,-2800,-775,-33428,775
C03132=-4946,57786,-1400,-775,-33428,775
C03133=-4452,57760,-1434,-841,-33411,577
C03134=-4452,57760,-2834,-841,-33411,577
C03135=-4413,57758,-2837,-847,-33410,562
C03136=-4413,57758,-1437,-847,-33410,562
C03137=-3784,57725,-1480,-931,-33389,310
C03138=-3784,57725,-2880,-931,-33389,310
C03139=-3692,57720,-2886,-943,-33386,274
C03140=-3692,57720,-1486,-943,-33386,274
C03141=-5049,57747,-1460,-762,-33404,817
C03142=-5049,57747,-2860,-762,-33404,817
C03143=-4989,57744,-2864,-770,-33402,793
C03144=-4989,57744,-1464,-770,-33402,793
C03145=-4449,57715,-1501,-842,-33384,577
C03146=-4449,57715,-2901,-842,-33384,577
C03147=-4407,57713,-2904,-848,-33383,560
C03148=-4407,57713,-1504,-848,-33383,560
C03149=-3746,57678,-1549,-936,-33361,296
C03150=-3746,57678,-2949,-936,-33361,296
C03151=-3654,57673,-2956,-949,-33358,259
C03152=-3654,57673,-1556,-949,-33358,259
C03153=-5089,57704,-1525,-757,-33379,834
C03154=-5089,57704,-2925,-757,-33379,834
C03155=-5033,57701,-2928,-765,-33377,811
C03156=-5033,57701,-1528,-765,-33377,811
C03157=-4446,57671,-1569,-843,-33357,576
C03158=-4446,57671,-2969,-843,-33357,576
C03159=-4404,57668,-2971,-849,-33356,559
C03160=-4404,57668,-1571,-849,-33356,559
C03161=-3708,57632,-1619,-942,-33333,281
C03162=-3708,57632,-3019,-942,-33333,281
C03163=-3623,57627,-3025,-953,-33330,247
C03164=-3623,57627,-1625,-953,-33330,247
C03165=-5125,57662,-1589,-753,-33353,849
C03166=-5125,57662,-2989,-753,-33353,849
C03167=-5069,57659,-2993,-761,-33351,826
C03168=-5069,57659,-1593,-761,-33351,826
C03169=-4447,57626,-1636,-844,-33330,577
C03170=-4447,57626,-3036,-844,-33330,577
C03171=-4405,57624,-3038,-850,-33329,560
C03172=-4405,57624,-1638,-850,-33329,560
C03173=-3674,57586,-1688,-947,-33304,268
C03174=-3674,57586,-3088,-947,-33304,268
C03175=-3578,57581,-3095,-960,-33301,230
C03176=-3578,57581,-1695,-960,-33301,230
C03177=-5165,57619,-1654,-748,-33328,865
C03178=-5165,57619,-3054,-748,-33328,865
C03179=-5105,57616,-3058,-757,-33326,841
C03180=-5105,57616,-1658,-757,-33326,841
C03181=-4445,57582,-1703,-845,-33303,577
C03182=-4445,57582,-3103,-845,-33303,577
C03183=-4402,57580,-3106,-851,-33302,560
C03184=-4402,57580,-1706,-851,-33302,560
C03185=-3650,57540,-1757,-951,-33277,259
C03186=-3650,57540,-3157,-951,-33277,259
C03187=-3590,57537,-3161,-959,-33275,235
C03188=-3590,57537,-1761,-959,-33275,235
C03189=-5202,57577,-1718,-744,-33302,880
C03190=-5202,57577,-3118,-744,-33302,880
C03191=-5138,57574,-3122,-753,-33300,855
C03192=-5138,57574,-1722,-753,-33300,855
C03193=-4442,57537,-1770,-846,-33276,576
C03194=-4442,57537,-3170,-846,-33276,576
C03195=-4407,57535,-3172,-851,-33275,562
C03196=-4407,57535,-1772,-851,-33275,562
C03197=-3676,57497,-1822,-949,-33251,270
C03198=-3676,57497,-3222,-949,-33251,270
C03199=-3608,57494,-3227,-958,-33248,243
C03200=-3608,57494,-1827,-958,-33248,243
C03201=-5231,57534,-1783,-741,-33276,892
C03202=-5231,57534,-3183,-741,-33276,892
C03203=-5178,57531,-3187,-748,-33274,871
C03204=-5178,57531,-1787,-748,-33274,871
C03205=-4443,57493,-1837,-847,-33249,577
C03206=-4443,57493,-3237,-847,-33249,577
C03207=-4401,57491,-3240,-852,-33248,560
C03208=-4401,57491,-1840,-852,-33248,560
C03209=-3701,57454,-1888,-946,-33224,281
C03210=-3701,57454,-3288,-946,-33224,281
C03211=-3631,57450,-3293,-955,-33222,252
C03212=-3631,57450,-1893,-955,-33222,252
C03213=-5264,57491,-1848,-737,-33250,906
C03214=-5264,57491,-3248,-737,-33250,906
C03215=-5211,57488,-3252,-744,-33248,885
C03216=-5211,57488,-1852,-744,-33248,885
C03217=-4444,57448,-1904,-847,-33222,578
C03218=-4444,57448,-3304,-847,-33222,578
C03219=-4402,57446,-3307,-853,-33221,561
C03220=-4402,57446,-1907,-853,-33221,561
C03221=-3734,57411,-1953,-942,-33198,294
C03222=-3734,57411,-3353,-942,-33198,294
C03223=-3660,57408,-3358,-952,-33196,265
C03224=-3660,57408,-1958,-952,-33196,265
C03225=-5300,57449,-1913,-733,-33224,921
C03226=-5300,57449,-3313,-733,-33224,921
C03227=-5240,57445,-3317,-741,-33222,897
C03228=-5240,57445,-1917,-741,-33222,897
C03229=-4441,57404,-1971,-848,-33195,578
C03230=-4441,57404,-3371,-848,-33195,578
C03231=-4399,57402,-3374,-854,-33194,561
C03232=-4399,57402,-1974,-854,-33194,561
C03233=-3763,57369,-2018,-939,-33172,306
C03234=-3763,57369,-3418,-939,-33172,306
C03235=-3696,57365,-3422,-948,-33170,280
C03236=-3696,57365,-2022,-948,-33170,280
C03237=-5333,57406,-1977,-729,-33198,935
C03238=-5333,57406,-3377,-729,-33198,935
C03239=-5269,57402,-3382,-738,-33196,909
C03240=-5269,57402,-1982,-738,-33196,909
C03241=-4439,57359,-2039,-849,-33168,577
C03242=-4439,57359,-3439,-849,-33168,577
C03243=-4396,57357,-3441,-855,-33167,560
C03244=-4396,57357,-2041,-855,-33167,560
C03245=-3803,57326,-2082,-934,-33147,323
C03246=-3803,57326,-3482,-934,-33147,323
C03247=-3736,57323,-3487,-943,-33145,296
C03248=-3736,57323,-2087,-943,-33145,296
C03249=-5366,57363,-2042,-726,-33173,948
C03250=-5366,57363,-3442,-726,-33173,948
C03251=-5302,57360,-3447,-734,-33171,923
C03252=-5302,57360,-2047,-734,-33171,923
C03253=-4440,57315,-2106,-850,-33141,578
C03254=-4440,57315,-3506,-850,-33141,578
C03255=-4397,57313,-3508,-855,-33140,561
C03256=-4397,57313,-2108,-855,-33140,561
C03257=-3836,57284,-2147,-931,-33121,337
C03258=-3836,57284,-3547,-931,-33121,337
C03259=-3776,57281,-3551,-939,-33119,313
C03260=-3776,57281,-2151,-939,-33119,313
C03261=-5381,57319,-2108,-724,-33146,955
C03262=-5381,57319,-3508,-724,-33146,955
C03263=-5275,57314,-3516,-738,-33143,912
C03264=-5275,57314,-2116,-738,-33143,912
C03265=-4441,57271,-2173,-850,-33114,579
C03266=-4441,57271,-3573,-850,-33114,579
C03267=-4398,57268,-3575,-856,-33113,562
C03268=-4398,57268,-2175,-856,-33113,562
C03269=-3872,57241,-2211,-926,-33095,352
C03270=-3872,57241,-3611,-926,-33095,352
C03271=-3812,57238,-3615,-935,-33093,328
C03272=-3812,57238,-2215,-935,-33093,328
C03273=-5346,57273,-2178,-730,-33118,942
C03274=-5346,57273,-3578,-730,-33118,942
C03275=-5233,57267,-3586,-745,-33114,896
C03276=-5233,57267,-2186,-745,-33114,896
C03277=-4438,57226,-2240,-851,-33087,579
C03278=-4438,57226,-3640,-851,-33087,579
C03279=-4396,57224,-3643,-857,-33086,562
C03280=-4396,57224,-2243,-857,-33086,562
C03281=-3905,57199,-2276,-923,-33069,365
C03282=-3905,57199,-3676,-923,-33069,365
C03283=-3852,57196,-3680,-930,-33067,344
C03284=-3852,57196,-2280,-930,-33067,344
C03285=-5284,57225,-2249,-739,-33089,917
C03286=-5284,57225,-3649,-739,-33089,917
C03287=-5181,57220,-3656,-752,-33086,876
C03288=-5181,57220,-2256,-752,-33086,876
C03289=-4439,57182,-2307,-852,-33060,579
C03290=-4439,57182,-3707,-852,-33060,579
C03291=-4397,57180,-3710,-857,-33059,562
C03292=-4397,57180,-2310,-857,-33059,562
C03293=-3948,57156,-2340,-918,-33044,383
C03294=-3948,57156,-3740,-918,-33044,383
C03295=-3884,57153,-3745,-926,-33042,358
C03296=-3884,57153,-2345,-926,-33042,358
C03297=-5228,57178,-2320,-747,-33060,895
C03298=-5228,57178,-3720,-747,-33060,895
C03299=-5126,57173,-3727,-760,-33057,854
C03300=-5126,57173,-2327,-760,-33057,854
C03301=-4437,57137,-2374,-853,-33033,579
C03302=-4437,57137,-3774,-853,-33033,579
C03303=-4398,57135,-3777,-858,-33032,563
C03304=-4398,57135,-2377,-858,-33032,563
C03305=-3991,57114,-2404,-913,-33018,401
C03306=-3991,57114,-3804,-913,-33018,401
C03307=-3928,57111,-3809,-921,-33016,376
C03308=-3928,57111,-2409,-921,-33016,376
C03309=-5169,57130,-2391,-755,-33031,872
C03310=-5169,57130,-3791,-755,-33031,872
C03311=-5067,57125,-3798,-769,-33028,831
C03312=-5067,57125,-2398,-769,-33028,831
C03313=-4434,57093,-2441,-854,-33006,578
C03314=-4434,57093,-3841,-854,-33006,578
C03315=-4399,57091,-3844,-859,-33005,564
C03316=-4399,57091,-2444,-859,-33005,564
C03317=-4038,57072,-2468,-907,-32993,420
C03318=-4038,57072,-3868,-907,-32993,420
C03319=-3971,57069,-3873,-916,-32991,393
C03320=-3971,57069,-2473,-916,-32991,393
C03321=-5114,57083,-2462,-763,-33002,851
C03322=-5114,57083,-3862,-763,-33002,851
C03323=-5000,57077,-3870,-779,-32999,805
C03324=-5000,57077,-2470,-779,-32999,805
C03325=-4435,57048,-2508,-854,-32979,579
C03326=-4435,57048,-3908,-854,-32979,579
C03327=-4396,57046,-3911,-860,-32978,564
C03328=-4396,57046,-2511,-860,-32978,564
C03329=-4081,57030,-2532,-902,-32967,438
C03330=-4081,57030,-3932,-902,-32967,438
C03331=-4021,57027,-3936,-910,-32965,414
C03332=-4021,57027,-2536,-910,-32965,414
C03333=-5058,57036,-2533,-772,-32974,829
C03334=-5058,57036,-3933,-772,-32974,829
C03335=-4938,57030,-3941,-788,-32970,781
C03336=-4938,57030,-2541,-788,-32970,781
C03337=-4436,57004,-2575,-855,-32952,580
C03338=-4436,57004,-3975,-855,-32952,580
C03339=-4397,57002,-3978,-860,-32951,565
C03340=-4397,57002,-2578,-860,-32951,565
C03341=-4125,56988,-2597,-897,-32942,456
C03342=-4125,56988,-3997,-897,-32942,456
C03343=-4058,56985,-4001,-906,-32940,429
C03344=-4058,56985,-2601,-906,-32940,429
C03345=-4985,56988,-2605,-782,-32944,800
C03346=-4985,56988,-4005,-782,-32944,800
C03347=-4872,56982,-4013,-797,-32940,755
C03348=-4872,56982,-2613,-797,-32940,755
C03349=-4437,56960,-2642,-856,-32925,581
C03350=-4437,56960,-4042,-856,-32925,581
C03351=-4398,56958,-4045,-861,-32924,566
C03352=-4398,56958,-2645,-861,-32924,566
C03353=-4168,56946,-2661,-892,-32916,474
C03354=-4168,56946,-4061,-892,-32916,474
C03355=-4097,56942,-4065,-901,-32914,446
C03356=-4097,56942,-2665,-901,-32914,446
C03357=-4915,56940,-2677,-792,-32915,773
C03358=-4915,56940,-4077,-792,-32915,773
C03359=-4791,56933,-4085,-809,-32911,723
C03360=-4791,56933,-2685,-809,-32911,723
C03361=-4438,56915,-2709,-856,-32899,582
C03362=-4438,56915,-4109,-856,-32899,582
C03363=-4399,56913,-4112,-861,-32897,567
C03364=-4399,56913,-2712,-861,-32897,567
C03365=-4204,56903,-2725,-887,-32891,489
C03366=-4204,56903,-4125,-887,-32891,489
C03367=-4144,56900,-4129,-895,-32889,465
C03368=-4144,56900,-2729,-895,-32889,465
C03369=-4852,56892,-2748,-801,-32886,748
C03370=-4852,56892,-4148,-801,-32886,748
C03371=-4722,56885,-4157,-819,-32881,696
C03372=-4722,56885,-2757,-819,-32881,696
C03373=-4439,56871,-2776,-857,-32872,583
C03374=-4439,56871,-4176,-857,-32872,583
C03375=-4400,56869,-4179,-862,-32870,567
C03376=-4400,56869,-2779,-862,-32870,567
C03377=-4237,56861,-2790,-884,-32865,503
C03378=-4237,56861,-4190,-884,-32865,503
C03379=-4177,56857,-4194,-892,-32863,478
C03380=-4177,56857,-2794,-892,-32863,478
C03381=-4776,56844,-2820,-812,-32856,718
C03382=-4776,56844,-4220,-812,-32856,718
C03383=-4655,56837,-4229,-828,-32852,670
C03384=-4655,56837,-2829,-828,-32852,670
C03385=-4440,56826,-2843,-857,-32845,584
C03386=-4440,56826,-4243,-857,-32845,584
C03387=-4401,56824,-4246,-862,-32843,568
C03388=-4401,56824,-2846,-862,-32843,568
C03389=-4273,56818,-2855,-879,-32839,518
C03390=-4273,56818,-4255,-879,-32839,518
C03391=-4210,56815,-4259,-888,-32837,492
C03392=-4210,56815,-2859,-888,-32837,492
C03393=-4706,56796,-2892,-822,-32827,691
C03394=-4706,56796,-4292,-822,-32827,691
C03395=-4600,56790,-4300,-836,-32823,648
C03396=-4600,56790,-2900,-836,-32823,648
C03397=-4441,56782,-2910,-858,-32818,585
C03398=-4441,56782,-4310,-858,-32818,585
C03399=-4398,56780,-4313,-863,-32816,568
C03400=-4398,56780,-2913,-863,-32816,568
C03401=-4310,56775,-2919,-875,-32813,533
C03402=-4310,56775,-4319,-875,-32813,533
C03403=-4250,56772,-4323,-883,-32811,509
C03404=-4250,56772,-2923,-883,-32811,509
C03405=-4647,56748,-2963,-831,-32798,668
C03406=-4647,56748,-4363,-831,-32798,668
C03407=-4548,56743,-4370,-844,-32794,628
C03408=-4548,56743,-2970,-844,-32794,628
C03409=-4438,56738,-2978,-859,-32791,584
C03410=-4438,56738,-4378,-859,-32791,584
C03411=-4399,56736,-4380,-864,-32789,569
C03412=-4399,56736,-2980,-864,-32789,569
C03413=-4335,56732,-2985,-873,-32787,543
C03414=-4335,56732,-4385,-873,-32787,543
C03415=-4279,56729,-4388,-880,-32785,521
C03416=-4279,56729,-2988,-880,-32785,521
C03417=-4598,56701,-3034,-838,-32769,649
C03418=-4598,56701,-4434,-838,-32769,649
C03419=-4492,56696,-4441,-852,-32766,606
C03420=-4492,56696,-3041,-852,-32766,606
C03421=-4439,56693,-3045,-859,-32764,585
C03422=-4439,56693,-4445,-859,-32764,585
C03423=-4397,56691,-4447,-865,-32762,568
C03424=-4397,56691,-3047,-865,-32762,568
C03425=-4372,56690,-3049,-868,-32761,558
C03426=-4372,56690,-4449,-868,-32761,558
C03427=-4308,56687,-4454,-877,-32759,533
C03428=-4308,56687,-3054,-877,-32759,533
C03429=-4557,56655,-3104,-844,-32741,633
C03430=-4557,56655,-4504,-844,-32741,633
C03431=-4320,56643,-4520,-876,-32733,538
C03432=-4320,56643,-3120,-876,-32733,538
C03433=-4505,56608,-3174,-852,-32712,613
C03434=-4505,56608,-4574,-852,-32712,613
C03435=-4338,56599,-4586,-874,-32706,546
C03436=-4338,56599,-3186,-874,-32706,546
C03437=-4488,56562,-3242,-855,-32685,606
C03438=-4488,56562,-4642,-855,-32685,606
C03439=-4237,56550,-4660,-889,-32676,506
C03440=-4237,56550,-3260,-889,-32676,506
C03441=-4531,56520,-3307,-850,-32659,624
C03442=-4531,56520,-4707,-850,-32659,624
C03443=-4064,56497,-4738,-912,-32643,438
C03444=-4064,56497,-3338,-912,-32643,438
C03445=-4578,56478,-3370,-844,-32634,644
C03446=-4578,56478,-4770,-844,-32634,644
C03447=-4497,56474,-4776,-855,-32631,611
C03448=-4497,56474,-3376,-855,-32631,611
C03449=-4444,56471,-3380,-862,-32629,590
C03450=-4444,56471,-4780,-862,-32629,590
C03451=-4401,56469,-4783,-868,-32628,573
C03452=-4401,56469,-3383,-868,-32628,573
C03453=-4193,56459,-3397,-896,-32620,490
C03454=-4193,56459,-4797,-896,-32620,490
C03455=-3895,56444,-4817,-936,-32610,371
C03456=-3895,56444,-3417,-936,-32610,371
C03457=-4636,56437,-3434,-837,-32609,667
C03458=-4636,56437,-4834,-837,-32609,667
C03459=-4547,56432,-4840,-849,-32606,632
C03460=-4547,56432,-3440,-849,-32606,632
C03461=-4441,56427,-3447,-863,-32602,589
C03462=-4441,56427,-4847,-863,-32602,589
C03463=-4402,56425,-4850,-868,-32601,574
C03464=-4402,56425,-3450,-868,-32601,574
C03465=-4020,56406,-3475,-920,-32587,421
C03466=-4020,56406,-4875,-920,-32587,421
C03467=-3787,56394,-4891,-951,-32579,328
C03468=-3787,56394,-3491,-951,-32579,328
C03469=-4693,56395,-3497,-830,-32584,691
C03470=-4693,56395,-4897,-830,-32584,691
C03471=-4605,56391,-4903,-842,-32581,655
C03472=-4605,56391,-3503,-842,-32581,655
C03473=-4439,56382,-3514,-864,-32575,589
C03474=-4439,56382,-4914,-864,-32575,589
C03475=-4400,56380,-4917,-869,-32574,573
C03476=-4400,56380,-3517,-869,-32574,573
C03477=-3855,56353,-3554,-943,-32555,356
C03478=-3855,56353,-4954,-943,-32555,356
C03479=-3653,56343,-4967,-970,-32548,275
C03480=-3653,56343,-3567,-970,-32548,275
C03481=-4751,56353,-3560,-823,-32559,714
C03482=-4751,56353,-4960,-823,-32559,714
C03483=-4666,56349,-4966,-834,-32556,680
C03484=-4666,56349,-3566,-834,-32556,680
C03485=-4439,56338,-3581,-865,-32548,590
C03486=-4439,56338,-4981,-865,-32548,590
C03487=-4397,56336,-4984,-870,-32547,573
C03488=-4397,56336,-3584,-870,-32547,573
C03489=-3735,56303,-3629,-959,-32524,309
C03490=-3735,56303,-5029,-959,-32524,309
C03491=-3505,56291,-5045,-990,-32516,217
C03492=-3505,56291,-3645,-990,-32516,217
C03493=-4805,56312,-3623,-816,-32534,736
C03494=-4805,56312,-5023,-816,-32534,736
C03495=-4720,56307,-5029,-828,-32531,702
C03496=-4720,56307,-3629,-828,-32531,702
C03497=-4437,56293,-3648,-866,-32521,589
C03498=-4437,56293,-5048,-866,-32521,589
C03499=-4394,56291,-5051,-871,-32519,572
C03500=-4394,56291,-3651,-871,-32519,572
C03501=-3616,56252,-3704,-976,-32492,261
C03502=-3616,56252,-5104,-976,-32492,261
C03503=-3361,56240,-5121,-1010,-32484,160
C03504=-3361,56240,-3721,-1010,-32484,160
C03505=-4852,56270,-3687,-811,-32508,756
C03506=-4852,56270,-5087,-811,-32508,756
C03507=-4778,56266,-5092,-821,-32506,726
C03508=-4778,56266,-3692,-821,-32506,726
C03509=-4438,56249,-3715,-866,-32494,590
C03510=-4438,56249,-5115,-866,-32494,590
C03511=-4392,56247,-5119,-872,-32492,572
C03512=-4392,56247,-3719,-872,-32492,572
C03513=-3472,56201,-3781,-996,-32460,204
C03514=-3472,56201,-5181,-996,-32460,204
C03515=-3344,56195,-5190,-1013,-32456,154
C03516=-3344,56195,-3790,-1013,-32456,154
C03517=-4913,56228,-3750,-803,-32484,781
C03518=-4913,56228,-5150,-803,-32484,781
C03519=-4832,56224,-5156,-814,-32481,748
C03520=-4832,56224,-3756,-814,-32481,748
C03521=-4439,56205,-3782,-867,-32467,591
C03522=-4439,56205,-5182,-867,-32467,591
C03523=-4396,56203,-5185,-873,-32466,574
C03524=-4396,56203,-3785,-873,-32466,574
C03525=-3402,56153,-3853,-1006,-32431,177
C03526=-3402,56153,-5253,-1006,-32431,177
C03527=-3345,56150,-5257,-1014,-32429,154
C03528=-3345,56150,-3857,-1014,-32429,154
C03529=-4971,56187,-3813,-796,-32459,804
C03530=-4971,56187,-5213,-796,-32459,804
C03531=-4889,56183,-5219,-807,-32456,772
C03532=-4889,56183,-3819,-807,-32456,772
C03533=-4436,56160,-3850,-868,-32440,591
C03534=-4436,56160,-5250,-868,-32440,591
C03535=-4390,56158,-5253,-874,-32438,572
C03536=-4390,56158,-3853,-874,-32438,572
C03537=-5021,56145,-3877,-790,-32433,825
C03538=-5021,56145,-5277,-790,-32433,825
C03539=-4947,56141,-5282,-800,-32431,795
C03540=-4947,56141,-3882,-800,-32431,795
C03541=-4434,56116,-3917,-869,-32413,590
C03542=-4434,56116,-5317,-869,-32413,590
C03543=-4395,56114,-5320,-874,-32412,575
C03544=-4395,56114,-3920,-874,-32412,575
C03545=-5082,56103,-3940,-782,-32409,850
C03546=-5082,56103,-5340,-782,-32409,850
C03547=-4994,56099,-5346,-794,-32406,814
C03548=-4994,56099,-3946,-794,-32406,814
C03549=-4435,56071,-3984,-869,-32386,591
C03550=-4435,56071,-5384,-869,-32386,591
C03551=-4392,56069,-5387,-875,-32385,574
C03552=-4392,56069,-3987,-875,-32385,574
C03553=-5143,56062,-4003,-775,-32384,875
C03554=-5143,56062,-5403,-775,-32384,875
C03555=-5055,56057,-5409,-787,-32381,839
C03556=-5055,56057,-4009,-787,-32381,839
C03557=-4432,56027,-4051,-870,-32359,591
C03558=-4432,56027,-5451,-870,-32359,591
C03559=-4393,56025,-5454,-876,-32358,575
C03560=-4393,56025,-4054,-876,-32358,575
C03561=-5215,56021,-4065,-766,-32359,904
C03562=-5215,56021,-5465,-766,-32359,904
C03563=-5113,56016,-5472,-780,-32356,863
C03564=-5113,56016,-4072,-780,-32356,863
C03565=-4433,55982,-4118,-871,-32332,591
C03566=-4433,55982,-5518,-871,-32332,591
C03567=-4387,55980,-5521,-877,-32330,573
C03568=-4387,55980,-4121,-877,-32330,573
C03569=-5269,55979,-4128,-759,-32334,926
C03570=-5269,55979,-5528,-759,-32334,926
C03571=-5170,55974,-5535,-772,-32331,886
C03572=-5170,55974,-4135,-772,-32331,886
C03573=-4430,55938,-4185,-872,-32305,591
C03574=-4430,55938,-5585,-872,-32305,591
C03575=-4388,55936,-5588,-878,-32303,574
C03576=-4388,55936,-4188,-878,-32303,574
C03577=-5270,55935,-4196,-760,-32308,927
C03578=-5270,55935,-5596,-760,-32308,927
C03579=-5217,55932,-5599,-767,-32306,906
C03580=-5217,55932,-4199,-767,-32306,906
C03581=-4435,55894,-4252,-872,-32278,593
C03582=-4435,55894,-5652,-872,-32278,593
C03583=-4385,55891,-5656,-879,-32276,574
C03584=-4385,55891,-4256,-879,-32276,574
C03585=-4432,55849,-4319,-873,-32251,593
C03586=-4432,55849,-5719,-873,-32251,593
C03587=-4390,55847,-5722,-879,-32250,576
C03588=-4390,55847,-4322,-879,-32250,576
C03589=-4433,55805,-4386,-874,-32224,594
C03590=-4433,55805,-5786,-874,-32224,594
C03591=-4345,55800,-5792,-886,-32221,558
C03592=-4345,55800,-4392,-886,-32221,558
C03593=-4438,55760,-4453,-874,-32197,596
C03594=-4438,55760,-5853,-874,-32197,596
C03595=-4335,55755,-5860,-888,-32194,555
C03596=-4335,55755,-4460,-888,-32194,555
C03597=-4439,55716,-4520,-874,-32170,597
C03598=-4439,55716,-5920,-874,-32170,597
C03599=-4329,55711,-5928,-889,-32166,553
C03600=-4329,55711,-4528,-889,-32166,553
C03601=-4450,55672,-4586,-873,-32144,602
C03602=-4450,55672,-5986,-873,-32144,602
C03603=-4319,55666,-5995,-891,-32139,550
C03604=-4319,55666,-4595,-891,-32139,550
C03605=-4444,55628,-4654,-875,-32117,600
C03606=-4444,55628,-6054,-875,-32117,600
C03607=-4313,55621,-6063,-893,-32112,548
C03608=-4313,55621,-4663,-893,-32112,548
C03609=-4452,55584,-4720,-875,-32090,604
C03610=-4452,55584,-6120,-875,-32090,604
C03611=-4378,55580,-6126,-885,-32087,574
C03612=-4378,55580,-4726,-885,-32087,574
C03613=-4360,55579,-4727,-887,-32087,567
C03614=-4360,55579,-6127,-887,-32087,567
C03615=-4303,55576,-6131,-895,-32085,545
C03616=-4303,55576,-4731,-895,-32085,545
C03617=-4456,55539,-4787,-875,-32063,606
C03618=-4456,55539,-6187,-875,-32063,606
C03619=-4400,55537,-6191,-882,-32061,584
C03620=-4400,55537,-4791,-882,-32061,584
C03621=-4347,55534,-4795,-889,-32059,562
C03622=-4347,55534,-6195,-889,-32059,562
C03623=-4290,55531,-6199,-897,-32057,540
C03624=-4290,55531,-4799,-897,-32057,540
C03625=-4465,55495,-4854,-874,-32036,610
C03626=-4465,55495,-6254,-874,-32036,610
C03627=-4415,55493,-6257,-881,-32035,590
C03628=-4415,55493,-4857,-881,-32035,590
C03629=-4337,55489,-4862,-891,-32032,559
C03630=-4337,55489,-6262,-891,-32032,559
C03631=-4280,55486,-6266,-899,-32030,537
C03632=-4280,55486,-4866,-899,-32030,537
C03633=-4473,55451,-4920,-874,-32010,614
C03634=-4473,55451,-6320,-874,-32010,614
C03635=-4427,55449,-6323,-880,-32008,595
C03636=-4427,55449,-4923,-880,-32008,595
C03637=-4324,55444,-4930,-894,-32004,554
C03638=-4324,55444,-6330,-894,-32004,554
C03639=-4267,55441,-6334,-902,-32002,532
C03640=-4267,55441,-4934,-902,-32002,532
C03641=-4484,55407,-4987,-873,-31983,619
C03642=-4484,55407,-6387,-873,-31983,619
C03643=-4438,55405,-6390,-879,-31982,601
C03644=-4438,55405,-4990,-879,-31982,601
C03645=-4307,55399,-4999,-897,-31977,548
C03646=-4307,55399,-6399,-897,-31977,548
C03647=-4254,55396,-6402,-904,-31975,527
C03648=-4254,55396,-5002,-904,-31975,527
C03649=-4496,55364,-5053,-872,-31957,624
C03650=-4496,55364,-6453,-872,-31957,624
C03651=-4450,55361,-6456,-878,-31955,606
C03652=-4450,55361,-5056,-878,-31955,606
C03653=-4297,55354,-5066,-899,-31950,545
C03654=-4297,55354,-6466,-899,-31950,545
C03655=-4248,55352,-6470,-906,-31948,525
C03656=-4248,55352,-5070,-906,-31948,525
C03657=-4511,55320,-5119,-871,-31930,631
C03658=-4511,55320,-6519,-871,-31930,631
C03659=-4461,55318,-6522,-877,-31928,611
C03660=-4461,55318,-5122,-877,-31928,611
C03661=-4284,55309,-5134,-901,-31922,540
C03662=-4284,55309,-6534,-901,-31922,540
C03663=-4234,55307,-6538,-908,-31920,520
C03664=-4234,55307,-5138,-908,-31920,520
C03665=-4522,55276,-5185,-870,-31904,636
C03666=-4522,55276,-6585,-870,-31904,636
C03667=-4473,55274,-6589,-877,-31902,616
C03668=-4473,55274,-5189,-877,-31902,616
C03669=-4274,55264,-5202,-903,-31895,537
C03670=-4274,55264,-6602,-903,-31895,537
C03671=-4221,55262,-6606,-911,-31893,516
C03672=-4221,55262,-5206,-911,-31893,516
C03673=-4530,55232,-5252,-869,-31877,640
C03674=-4530,55232,-6652,-869,-31877,640
C03675=-4484,55230,-6655,-876,-31875,621
C03676=-4484,55230,-5255,-876,-31875,621
C03677=-4258,55219,-5270,-906,-31867,531
C03678=-4258,55219,-6670,-906,-31867,531
C03679=-4208,55217,-6674,-913,-31865,511
C03680=-4208,55217,-5274,-913,-31865,511
C03681=-4538,55188,-5318,-869,-31850,643
C03682=-4538,55188,-6718,-869,-31850,643
C03683=-4500,55186,-6721,-874,-31849,628
C03684=-4500,55186,-5321,-874,-31849,628
C03685=-4244,55174,-5338,-909,-31840,526
C03686=-4244,55174,-6738,-909,-31840,526
C03687=-4195,55172,-6741,-915,-31838,506
C03688=-4195,55172,-5341,-915,-31838,506
C03689=-4550,55144,-5385,-868,-31824,648
C03690=-4550,55144,-6785,-868,-31824,648
C03691=-4511,55142,-6787,-873,-31822,633
C03692=-4511,55142,-5387,-873,-31822,633
C03693=-4231,55129,-5406,-911,-31812,521
C03694=-4231,55129,-6806,-911,-31812,521
C03695=-4181,55127,-6809,-918,-31810,501
C03696=-4181,55127,-5409,-918,-31810,501
C03697=-4558,55100,-5451,-868,-31797,652
C03698=-4558,55100,-6851,-868,-31797,652
C03699=-4519,55098,-6854,-873,-31796,637
C03700=-4519,55098,-5454,-873,-31796,637
C03701=-4218,55084,-5474,-914,-31785,517
C03702=-4218,55084,-6874,-914,-31785,517
C03703=-4172,55082,-6877,-920,-31783,498
C03704=-4172,55082,-5477,-920,-31783,498
C03705=-4573,55056,-5517,-866,-31771,659
C03706=-4573,55056,-6917,-866,-31771,659
C03707=-4531,55054,-6920,-872,-31769,642
C03708=-4531,55054,-5520,-872,-31769,642
C03709=-4208,55039,-5542,-916,-31757,513
C03710=-4208,55039,-6942,-916,-31757,513
C03711=-4162,55037,-6945,-922,-31756,495
C03712=-4162,55037,-5545,-922,-31756,495
C03713=-4581,55012,-5584,-866,-31744,663
C03714=-4581,55012,-6984,-866,-31744,663
C03715=-4542,55011,-6986,-871,-31743,647
C03716=-4542,55011,-5586,-871,-31743,647
C03717=-4195,54994,-5610,-918,-31730,508
C03718=-4195,54994,-7010,-918,-31730,508
C03719=-4152,54992,-7013,-924,-31728,491
C03720=-4152,54992,-5613,-924,-31728,491
C03721=-4593,54969,-5650,-865,-31717,668
C03722=-4593,54969,-7050,-865,-31717,668
C03723=-4557,54967,-7052,-870,-31716,654
C03724=-4557,54967,-5652,-870,-31716,654
C03725=-4189,54949,-5677,-920,-31703,507
C03726=-4189,54949,-7077,-920,-31703,507
C03727=-4139,54947,-7081,-926,-31701,487
C03728=-4139,54947,-5681,-926,-31701,487
C03729=-4604,54925,-5716,-864,-31691,673
C03730=-4604,54925,-7116,-864,-31691,673
C03731=-4569,54923,-7119,-869,-31690,659
C03732=-4569,54923,-5719,-869,-31690,659
C03733=-4175,54904,-5745,-922,-31675,502
C03734=-4175,54904,-7145,-922,-31675,502
C03735=-4126,54902,-7149,-929,-31674,482
C03736=-4126,54902,-5749,-929,-31674,482
C03737=-4616,54881,-5783,-863,-31664,678
C03738=-4616,54881,-7183,-863,-31664,678
C03739=-4581,54879,-7185,-868,-31663,664
C03740=-4581,54879,-5785,-868,-31663,664
C03741=-4162,54859,-5813,-925,-31648,497
C03742=-4162,54859,-7213,-925,-31648,497
C03743=-4116,54857,-7216,-931,-31646,479
C03744=-4116,54857,-5816,-931,-31646,479
C03745=-4624,54837,-5849,-863,-31638,682
C03746=-4624,54837,-7249,-863,-31638,682
C03747=-4589,54835,-7251,-868,-31636,668
C03748=-4589,54835,-5851,-868,-31636,668
C03749=-4156,54815,-5881,-926,-31621,495
C03750=-4156,54815,-7281,-926,-31621,495
C03751=-4103,54812,-7284,-933,-31619,474
C03752=-4103,54812,-5884,-933,-31619,474
C03753=-4636,54793,-5915,-862,-31611,687
C03754=-4636,54793,-7315,-862,-31611,687
C03755=-4600,54791,-7318,-867,-31610,673
C03756=-4600,54791,-5918,-867,-31610,673
C03757=-4139,54770,-5949,-929,-31593,489
C03758=-4139,54770,-7349,-929,-31593,489
C03759=-4086,54767,-7352,-936,-31591,468
C03760=-4086,54767,-5952,-936,-31591,468
C03761=-4647,54749,-5982,-861,-31585,692
C03762=-4647,54749,-7382,-861,-31585,692
C03763=-4612,54747,-7384,-866,-31583,678
C03764=-4612,54747,-5984,-866,-31583,678
C03765=-4126,54725,-6017,-932,-31566,484
C03766=-4126,54725,-7417,-932,-31566,484
C03767=-4073,54722,-7420,-939,-31564,463
C03768=-4073,54722,-6020,-939,-31564,463
C03769=-4655,54705,-6048,-861,-31558,696
C03770=-4655,54705,-7448,-861,-31558,696
C03771=-4620,54703,-7451,-866,-31557,682
C03772=-4620,54703,-6051,-866,-31557,682
C03773=-4109,54679,-6085,-935,-31538,478
C03774=-4109,54679,-7485,-935,-31538,478
C03775=-4060,54677,-7488,-941,-31536,458
C03776=-4060,54677,-6088,-941,-31536,458
C03777=-4663,54661,-6115,-860,-31531,700
C03778=-4663,54661,-7515,-860,-31531,700
C03779=-4628,54659,-7517,-865,-31530,685
C03780=-4628,54659,-6117,-865,-31530,685
C03781=-4099,54635,-6153,-937,-31511,475
C03782=-4099,54635,-7553,-937,-31511,475
C03783=-4053,54632,-7556,-943,-31509,456
C03784=-4053,54632,-6156,-943,-31509,456
C03785=-4675,54617,-6181,-859,-31505,705
C03786=-4675,54617,-7581,-859,-31505,705
C03787=-4640,54615,-7583,-864,-31503,691
C03788=-4640,54615,-6183,-864,-31503,691
C03789=-4083,54589,-6221,-940,-31483,469
C03790=-4083,54589,-7621,-940,-31483,469
C03791=-4040,54587,-7624,-945,-31482,452
C03792=-4040,54587,-6224,-945,-31482,452
C03793=-4687,54573,-6247,-859,-31478,710
C03794=-4687,54573,-7647,-859,-31478,710
C03795=-4651,54571,-7650,-863,-31477,696
C03796=-4651,54571,-6250,-863,-31477,696
C03797=-4069,54544,-6289,-942,-31456,464
C03798=-4069,54544,-7689,-942,-31456,464
C03799=-4027,54542,-7692,-948,-31454,447
C03800=-4027,54542,-6292,-948,-31454,447
C03801=-4698,54529,-6314,-858,-31452,715
C03802=-4698,54529,-7714,-858,-31452,715
C03803=-4663,54528,-7716,-862,-31450,701
C03804=-4663,54528,-6316,-862,-31450,701
C03805=-4060,54500,-6357,-944,-31428,461
C03806=-4060,54500,-7757,-944,-31428,461
C03807=-4017,54498,-7759,-950,-31427,444
C03808=-4017,54498,-6359,-950,-31427,444
C03809=-4713,54485,-6380,-856,-31425,722
C03810=-4713,54485,-7780,-856,-31425,722
C03811=-4678,54484,-7782,-861,-31424,707
C03812=-4678,54484,-6382,-861,-31424,707
C03813=-4050,54455,-6424,-946,-31401,457
C03814=-4050,54455,-7824,-946,-31401,457
C03815=-4007,54453,-7827,-952,-31399,440
C03816=-4007,54453,-6427,-952,-31399,440
C03817=-4728,54442,-6446,-855,-31399,728
C03818=-4728,54442,-7846,-855,-31399,728
C03819=-4693,54440,-7848,-860,-31397,714
C03820=-4693,54440,-6448,-860,-31397,714
C03821=-4037,54410,-6492,-949,-31373,452
C03822=-4037,54410,-7892,-949,-31373,452
C03823=-3994,54408,-7895,-954,-31372,436
C03824=-3994,54408,-6495,-954,-31372,436
C03825=-4744,54398,-6512,-854,-31372,735
C03826=-4744,54398,-7912,-854,-31372,735
C03827=-4705,54396,-7914,-859,-31371,719
C03828=-4705,54396,-6514,-859,-31371,719
C03829=-4031,54365,-6560,-950,-31346,451
C03830=-4031,54365,-7960,-950,-31346,451
C03831=-3977,54363,-7963,-957,-31344,429
C03832=-3977,54363,-6563,-957,-31344,429
C03833=-4755,54354,-6578,-853,-31346,740
C03834=-4755,54354,-7978,-853,-31346,740
C03835=-4716,54352,-7981,-858,-31344,724
C03836=-4716,54352,-6581,-858,-31344,724
C03837=-4014,54320,-6628,-953,-31319,444
C03838=-4014,54320,-8028,-953,-31319,444
C03839=-3960,54317,-8032,-960,-31317,423
C03840=-3960,54317,-6632,-960,-31317,423
C03841=-4767,54310,-6644,-852,-31319,745
C03842=-4767,54310,-8044,-852,-31319,745
C03843=-4728,54308,-8047,-857,-31318,730
C03844=-4728,54308,-6647,-857,-31318,730
C03845=-3997,54275,-6696,-956,-31291,438
C03846=-3997,54275,-8096,-956,-31291,438
C03847=-3947,54273,-8099,-963,-31289,418
C03848=-3947,54273,-6699,-963,-31289,418
C03849=-4778,54266,-6711,-851,-31293,750
C03850=-4778,54266,-8111,-851,-31293,750
C03851=-4739,54265,-8113,-856,-31291,735
C03852=-4739,54265,-6713,-856,-31291,735
C03853=-3980,54230,-6764,-959,-31263,432
C03854=-3980,54230,-8164,-959,-31263,432
C03855=-3930,54227,-8168,-966,-31262,412
C03856=-3930,54227,-6768,-966,-31262,412
C03857=-4787,54222,-6777,-850,-31266,754
C03858=-4787,54222,-8177,-850,-31266,754
C03859=-4751,54221,-8180,-855,-31265,740
C03860=-4751,54221,-6780,-855,-31265,740
C03861=-3963,54185,-6833,-962,-31236,426
C03862=-3963,54185,-8233,-962,-31236,426
C03863=-3910,54182,-8236,-969,-31234,405
C03864=-3910,54182,-6836,-969,-31234,405
C03865=-4798,54178,-6843,-850,-31240,759
C03866=-4798,54178,-8243,-850,-31240,759
C03867=-4759,54177,-8246,-855,-31238,744
C03868=-4759,54177,-6846,-855,-31238,744
C03869=-3950,54140,-6900,-964,-31208,421
C03870=-3950,54140,-8300,-964,-31208,421
C03871=-3890,54137,-8305,-973,-31206,397
C03872=-3890,54137,-6905,-973,-31206,397
C03873=-4806,54134,-6910,-849,-31213,763
C03874=-4806,54134,-8310,-849,-31213,763
C03875=-4767,54133,-8313,-854,-31211,747
C03876=-4767,54133,-6913,-854,-31211,747
C03877=-3926,54094,-6969,-968,-31180,412
C03878=-3926,54094,-8369,-968,-31180,412
C03879=-3873,54092,-8373,-976,-31178,391
C03880=-3873,54092,-6973,-976,-31178,391
C03881=-4814,54090,-6977,-849,-31186,767
C03882=-4814,54090,-8377,-849,-31186,767
C03883=-4779,54089,-8379,-854,-31185,753
C03884=-4779,54089,-6979,-854,-31185,753
C03885=-3909,54049,-7037,-971,-31153,406
C03886=-3909,54049,-8437,-971,-31153,406
C03887=-3856,54047,-8441,-979,-31151,385
C03888=-3856,54047,-7041,-979,-31151,385
C03889=-4829,54047,-7043,-847,-31160,773
C03890=-4829,54047,-8443,-847,-31160,773
C03891=-4787,54045,-8445,-853,-31158,756
C03892=-4787,54045,-7045,-853,-31158,756
C03893=-3885,54004,-7106,-975,-31125,397
C03894=-3885,54004,-8506,-975,-31125,397
C03895=-3839,54001,-8509,-982,-31123,379
C03896=-3839,54001,-7109,-982,-31123,379
C03897=-4837,54002,-7109,-847,-31133,777
C03898=-4837,54002,-8509,-847,-31133,777
C03899=-4798,54001,-8512,-852,-31132,761
C03900=-4798,54001,-7112,-852,-31132,761
C03901=-3872,53959,-7174,-978,-31097,392
C03902=-3872,53959,-8574,-978,-31097,392
C03903=-3826,53956,-8577,-984,-31096,374
C03904=-3826,53956,-7177,-984,-31096,374
C03905=-4849,53959,-7175,-846,-31107,782
C03906=-4849,53959,-8575,-846,-31107,782
C03907=-4814,53957,-8578,-851,-31105,768
C03908=-4814,53957,-7178,-851,-31105,768
C03909=-3855,53913,-7242,-981,-31070,386
C03910=-3855,53913,-8642,-981,-31070,386
C03911=-3813,53911,-8645,-987,-31068,369
C03912=-3813,53911,-7245,-987,-31068,369
C03913=-4864,53915,-7241,-845,-31080,789
C03914=-4864,53915,-8641,-845,-31080,789
C03915=-4825,53913,-8644,-850,-31079,773
C03916=-4825,53913,-7244,-850,-31079,773
C03917=-3845,53869,-7310,-983,-31042,383
C03918=-3845,53869,-8710,-983,-31042,383
C03919=-3799,53867,-8713,-989,-31041,364
C03920=-3799,53867,-7313,-989,-31041,364
C03921=-4869,53871,-7308,-845,-31053,791
C03922=-4869,53871,-8708,-845,-31053,791
C03923=-4837,53869,-8710,-849,-31052,778
C03924=-4837,53869,-7310,-849,-31052,778
C03925=-3832,53824,-7378,-985,-31015,378
C03926=-3832,53824,-8778,-985,-31015,378
C03927=-3782,53821,-8781,-992,-31013,358
C03928=-3782,53821,-7381,-992,-31013,358
C03929=-4880,53827,-7375,-844,-31027,796
C03930=-4880,53827,-8775,-844,-31027,796
C03931=-4841,53825,-8777,-849,-31025,781
C03932=-4841,53825,-7377,-849,-31025,781
C03933=-3815,53779,-7446,-988,-30987,372
C03934=-3815,53779,-8846,-988,-30987,372
C03935=-3769,53776,-8849,-995,-30986,354
C03936=-3769,53776,-7449,-995,-30986,354
C03937=-4892,53783,-7441,-843,-31000,801
C03938=-4892,53783,-8841,-843,-31000,801
C03939=-4849,53781,-8844,-849,-30999,784
C03940=-4849,53781,-7444,-849,-30999,784
C03941=-3802,53734,-7514,-991,-30960,367
C03942=-3802,53734,-8914,-991,-30960,367
C03943=-3756,53732,-8917,-997,-30958,349
C03944=-3756,53732,-7517,-997,-30958,349
C03945=-4900,53739,-7507,-842,-30974,805
C03946=-4900,53739,-8907,-842,-30974,805
C03947=-4861,53737,-8910,-848,-30972,790
C03948=-4861,53737,-7510,-848,-30972,790
C03949=-3785,53689,-7582,-994,-30932,361
C03950=-3785,53689,-8982,-994,-30932,361
C03951=-3739,53686,-8985,-1000,-30930,343
C03952=-3739,53686,-7585,-1000,-30930,343
C03953=-4912,53695,-7574,-842,-30947,810
C03954=-4912,53695,-8974,-842,-30947,810
C03955=-4869,53693,-8977,-847,-30946,793
C03956=-4869,53693,-7577,-847,-30946,793
C03957=-3775,53644,-7650,-996,-30905,358
C03958=-3775,53644,-9050,-996,-30905,358
C03959=-3722,53641,-9053,-1003,-30903,336
C03960=-3722,53641,-7653,-1003,-30903,336
C03961=-4923,53651,-7640,-841,-30921,815
C03962=-4923,53651,-9040,-841,-30921,815
C03963=-4877,53649,-9043,-847,-30919,797
C03964=-4877,53649,-7643,-847,-30919,797
C03965=-3758,53599,-7718,-999,-30877,352
C03966=-3758,53599,-9118,-999,-30877,352
C03967=-3702,53596,-9122,-1006,-30875,329
C03968=-3702,53596,-7722,-1006,-30875,329
C03969=-4946,53607,-7706,-838,-30895,825
C03970=-4946,53607,-9106,-838,-30895,825
C03971=-4885,53605,-9110,-846,-30892,801
C03972=-4885,53605,-7710,-846,-30892,801
C03973=-3738,53553,-7786,-1002,-30849,344
C03974=-3738,53553,-9186,-1002,-30849,344
C03975=-3678,53551,-9191,-1010,-30847,320
C03976=-3678,53551,-7791,-1010,-30847,320
C03977=-4954,53563,-7772,-838,-30868,829
C03978=-4954,53563,-9172,-838,-30868,829
C03979=-4900,53561,-9176,-845,-30866,807
C03980=-4900,53561,-7776,-845,-30866,807
C03981=-3718,53508,-7855,-1006,-30822,336
C03982=-3718,53508,-9255,-1006,-30822,336
C03983=-3664,53506,-9258,-1013,-30820,315
C03984=-3664,53506,-7858,-1013,-30820,315
C03985=-4962,53519,-7839,-837,-30841,832
C03986=-4962,53519,-9239,-837,-30841,832
C03987=-4901,53517,-9243,-846,-30839,808
C03988=-4901,53517,-7843,-846,-30839,808
C03989=-3701,53463,-7923,-1009,-30794,330
C03990=-3701,53463,-9323,-1009,-30794,330
C03991=-3651,53461,-9326,-1015,-30792,310
C03992=-3651,53461,-7926,-1015,-30792,310
C03993=-4970,53475,-7905,-837,-30815,836
C03994=-4970,53475,-9305,-837,-30815,836
C03995=-4913,53473,-9309,-845,-30812,813
C03996=-4913,53473,-7909,-845,-30812,813
C03997=-3688,53418,-7991,-1011,-30766,325
C03998=-3688,53418,-9391,-1011,-30766,325
C03999=-3638,53416,-9394,-1018,-30765,306
C04000=-3638,53416,-7994,-1018,-30765,306
C04001=-4978,53431,-7972,-837,-30788,840
C04002=-4978,53431,-9372,-837,-30788,840
C04003=-4925,53429,-9375,-844,-30786,819
C04004=-4925,53429,-7975,-844,-30786,819
C04005=-3674,53373,-8059,-1014,-30739,321
C04006=-3674,53373,-9459,-1014,-30739,321
C04007=-3628,53371,-9462,-1020,-30737,302
C04008=-3628,53371,-8062,-1020,-30737,302
C04009=-4982,53387,-8038,-837,-30761,842
C04010=-4982,53387,-9438,-837,-30761,842
C04011=-4933,53385,-9442,-843,-30759,822
C04012=-4933,53385,-8042,-843,-30759,822
C04013=-3661,53328,-8127,-1016,-30711,316
C04014=-3661,53328,-9527,-1016,-30711,316
C04015=-3611,53326,-9530,-1023,-30710,296
C04016=-3611,53326,-8130,-1023,-30710,296
C04017=-4980,53342,-8106,-838,-30734,842
C04018=-4980,53342,-9506,-838,-30734,842
C04019=-4948,53341,-9508,-842,-30733,829
C04020=-4948,53341,-8108,-842,-30733,829
C04021=-3655,53284,-8194,-1018,-30684,314
C04022=-3655,53284,-9594,-1018,-30684,314
C04023=-3601,53281,-9598,-1025,-30682,293
C04024=-3601,53281,-8198,-1025,-30682,293
C04025=-3648,53239,-8262,-1019,-30657,312
C04026=-3648,53239,-9662,-1019,-30657,312
C04027=-3592,53237,-9666,-1027,-30655,290
C04028=-3592,53237,-8266,-1027,-30655,290
C04029=-3642,53194,-8329,-1021,-30630,310
C04030=-3642,53194,-9729,-1021,-30630,310
C04031=-3582,53192,-9733,-1029,-30627,286
C04032=-3582,53192,-8333,-1029,-30627,286
C04033=-3632,53150,-8397,-1023,-30602,307
C04034=-3632,53150,-9797,-1023,-30602,307
C04035=-3579,53147,-9801,-1030,-30600,286
C04036=-3579,53147,-8401,-1030,-30600,286
C04037=-3612,53104,-8466,-1026,-30575,299
C04038=-3612,53104,-9866,-1026,-30575,299
C04039=-3584,53103,-9867,-1030,-30573,288
C04040=-3584,53103,-8467,-1030,-30573,288
//INST
///DATE 2026/04/22 19:50
///ATTR SC,RW
///GROUP1 RB1
NOP
MOVJ C00000 VJ=0.78
MOVJ C00001 VJ=0.78
MOVJ C00002 VJ=0.78
MOVL C00003 V=8.0
MOVJ C00004 VJ=0.78
MOVJ C00005 VJ=0.78
MOVJ C00006 VJ=0.78
MOVL C00007 V=8.0
MOVJ C00008 VJ=0.78
MOVJ C00009 VJ=0.78
MOVJ C00010 VJ=0.78
MOVL C00011 V=8.0
MOVJ C00012 VJ=0.78
MOVJ C00013 VJ=0.78
MOVJ C00014 VJ=0.78
MOVL C00015 V=8.0
MOVJ C00016 VJ=0.78
MOVJ C00017 VJ=0.78
MOVJ C00018 VJ=0.78
MOVL C00019 V=8.0
MOVJ C00020 VJ=0.78
MOVJ C00021 VJ=0.78
MOVJ C00022 VJ=0.78
MOVL C00023 V=8.0
MOVJ C00024 VJ=0.78
MOVJ C00025 VJ=0.78
MOVJ C00026 VJ=0.78
MOVL C00027 V=8.0
MOVJ C00028 VJ=0.78
MOVJ C00029 VJ=0.78
MOVJ C00030 VJ=0.78
MOVL C00031 V=8.0
MOVJ C00032 VJ=0.78
MOVJ C00033 VJ=0.78
MOVJ C00034 VJ=0.78
MOVL C00035 V=8.0
MOVJ C00036 VJ=0.78
MOVJ C00037 VJ=0.78
MOVJ C00038 VJ=0.78
MOVL C00039 V=8.0
MOVJ C00040 VJ=0.78
MOVJ C00041 VJ=0.78
MOVJ C00042 VJ=0.78
MOVL C00043 V=8.0
MOVJ C00044 VJ=0.78
MOVJ C00045 VJ=0.78
MOVJ C00046 VJ=0.78
MOVL C00047 V=8.0
MOVJ C00048 VJ=0.78
MOVJ C00049 VJ=0.78
MOVJ C00050 VJ=0.78
MOVL C00051 V=8.0
MOVJ C00052 VJ=0.78
MOVJ C00053 VJ=0.78
MOVJ C00054 VJ=0.78
MOVL C00055 V=8.0
MOVJ C00056 VJ=0.78
MOVJ C00057 VJ=0.78
MOVJ C00058 VJ=0.78
MOVL C00059 V=8.0
MOVJ C00060 VJ=0.78
MOVJ C00061 VJ=0.78
MOVJ C00062 VJ=0.78
MOVL C00063 V=8.0
MOVJ C00064 VJ=0.78
MOVJ C00065 VJ=0.78
MOVJ C00066 VJ=0.78
MOVL C00067 V=8.0
MOVJ C00068 VJ=0.78
MOVJ C00069 VJ=0.78
MOVJ C00070 VJ=0.78
MOVL C00071 V=8.0
MOVJ C00072 VJ=0.78
MOVJ C00073 VJ=0.78
MOVJ C00074 VJ=0.78
MOVL C00075 V=8.0
MOVJ C00076 VJ=0.78
MOVJ C00077 VJ=0.78
MOVJ C00078 VJ=0.78
MOVL C00079 V=8.0
MOVJ C00080 VJ=0.78
MOVJ C00081 VJ=0.78
MOVJ C00082 VJ=0.78
MOVL C00083 V=8.0
MOVJ C00084 VJ=0.78
MOVJ C00085 VJ=0.78
MOVJ C00086 VJ=0.78
MOVL C00087 V=8.0
MOVJ C00088 VJ=0.78
MOVJ C00089 VJ=0.78
MOVJ C00090 VJ=0.78
MOVL C00091 V=8.0
MOVJ C00092 VJ=0.78
MOVJ C00093 VJ=0.78
MOVJ C00094 VJ=0.78
MOVL C00095 V=8.0
MOVJ C00096 VJ=0.78
MOVJ C00097 VJ=0.78
MOVJ C00098 VJ=0.78
MOVL C00099 V=8.0
MOVJ C00100 VJ=0.78
MOVJ C00101 VJ=0.78
MOVJ C00102 VJ=0.78
MOVL C00103 V=8.0
MOVJ C00104 VJ=0.78
MOVJ C00105 VJ=0.78
MOVJ C00106 VJ=0.78
MOVL C00107 V=8.0
MOVJ C00108 VJ=0.78
MOVJ C00109 VJ=0.78
MOVJ C00110 VJ=0.78
MOVL C00111 V=8.0
MOVJ C00112 VJ=0.78
MOVJ C00113 VJ=0.78
MOVJ C00114 VJ=0.78
MOVL C00115 V=8.0
MOVJ C00116 VJ=0.78
MOVJ C00117 VJ=0.78
MOVJ C00118 VJ=0.78
MOVL C00119 V=8.0
MOVJ C00120 VJ=0.78
MOVJ C00121 VJ=0.78
MOVJ C00122 VJ=0.78
MOVL C00123 V=8.0
MOVJ C00124 VJ=0.78
MOVJ C00125 VJ=0.78
MOVJ C00126 VJ=0.78
MOVL C00127 V=8.0
MOVJ C00128 VJ=0.78
MOVJ C00129 VJ=0.78
MOVJ C00130 VJ=0.78
MOVL C00131 V=8.0
MOVJ C00132 VJ=0.78
MOVJ C00133 VJ=0.78
MOVJ C00134 VJ=0.78
MOVL C00135 V=8.0
MOVJ C00136 VJ=0.78
MOVJ C00137 VJ=0.78
MOVJ C00138 VJ=0.78
MOVL C00139 V=8.0
MOVJ C00140 VJ=0.78
MOVJ C00141 VJ=0.78
MOVJ C00142 VJ=0.78
MOVL C00143 V=8.0
MOVJ C00144 VJ=0.78
MOVJ C00145 VJ=0.78
MOVJ C00146 VJ=0.78
MOVL C00147 V=8.0
MOVJ C00148 VJ=0.78
MOVJ C00149 VJ=0.78
MOVJ C00150 VJ=0.78
MOVL C00151 V=8.0
MOVJ C00152 VJ=0.78
MOVJ C00153 VJ=0.78
MOVJ C00154 VJ=0.78
MOVL C00155 V=8.0
MOVJ C00156 VJ=0.78
MOVJ C00157 VJ=0.78
MOVJ C00158 VJ=0.78
MOVL C00159 V=8.0
MOVJ C00160 VJ=0.78
MOVJ C00161 VJ=0.78
MOVJ C00162 VJ=0.78
MOVL C00163 V=8.0
MOVJ C00164 VJ=0.78
MOVJ C00165 VJ=0.78
MOVJ C00166 VJ=0.78
MOVL C00167 V=8.0
MOVJ C00168 VJ=0.78
MOVJ C00169 VJ=0.78
MOVJ C00170 VJ=0.78
MOVL C00171 V=8.0
MOVJ C00172 VJ=0.78
MOVJ C00173 VJ=0.78
MOVJ C00174 VJ=0.78
MOVL C00175 V=8.0
MOVJ C00176 VJ=0.78
MOVJ C00177 VJ=0.78
MOVJ C00178 VJ=0.78
MOVL C00179 V=8.0
MOVJ C00180 VJ=0.78
MOVJ C00181 VJ=0.78
MOVJ C00182 VJ=0.78
MOVL C00183 V=8.0
MOVJ C00184 VJ=0.78
MOVJ C00185 VJ=0.78
MOVJ C00186 VJ=0.78
MOVL C00187 V=8.0
MOVJ C00188 VJ=0.78
MOVJ C00189 VJ=0.78
MOVJ C00190 VJ=0.78
MOVL C00191 V=8.0
MOVJ C00192 VJ=0.78
MOVJ C00193 VJ=0.78
MOVJ C00194 VJ=0.78
MOVL C00195 V=8.0
MOVJ C00196 VJ=0.78
MOVJ C00197 VJ=0.78
MOVJ C00198 VJ=0.78
MOVL C00199 V=8.0
MOVJ C00200 VJ=0.78
MOVJ C00201 VJ=0.78
MOVJ C00202 VJ=0.78
MOVL C00203 V=8.0
MOVJ C00204 VJ=0.78
MOVJ C00205 VJ=0.78
MOVJ C00206 VJ=0.78
MOVL C00207 V=8.0
MOVJ C00208 VJ=0.78
MOVJ C00209 VJ=0.78
MOVJ C00210 VJ=0.78
MOVL C00211 V=8.0
MOVJ C00212 VJ=0.78
MOVJ C00213 VJ=0.78
MOVJ C00214 VJ=0.78
MOVL C00215 V=8.0
MOVJ C00216 VJ=0.78
MOVJ C00217 VJ=0.78
MOVJ C00218 VJ=0.78
MOVL C00219 V=8.0
MOVJ C00220 VJ=0.78
MOVJ C00221 VJ=0.78
MOVJ C00222 VJ=0.78
MOVL C00223 V=8.0
MOVJ C00224 VJ=0.78
MOVJ C00225 VJ=0.78
MOVJ C00226 VJ=0.78
MOVL C00227 V=8.0
MOVJ C00228 VJ=0.78
MOVJ C00229 VJ=0.78
MOVJ C00230 VJ=0.78
MOVL C00231 V=8.0
MOVJ C00232 VJ=0.78
MOVJ C00233 VJ=0.78
MOVJ C00234 VJ=0.78
MOVL C00235 V=8.0
MOVJ C00236 VJ=0.78
MOVJ C00237 VJ=0.78
MOVJ C00238 VJ=0.78
MOVL C00239 V=8.0
MOVJ C00240 VJ=0.78
MOVJ C00241 VJ=0.78
MOVJ C00242 VJ=0.78
MOVL C00243 V=8.0
MOVJ C00244 VJ=0.78
MOVJ C00245 VJ=0.78
MOVJ C00246 VJ=0.78
MOVL C00247 V=8.0
MOVJ C00248 VJ=0.78
MOVJ C00249 VJ=0.78
MOVJ C00250 VJ=0.78
MOVL C00251 V=8.0
MOVJ C00252 VJ=0.78
MOVJ C00253 VJ=0.78
MOVJ C00254 VJ=0.78
MOVL C00255 V=8.0
MOVJ C00256 VJ=0.78
MOVJ C00257 VJ=0.78
MOVJ C00258 VJ=0.78
MOVL C00259 V=8.0
MOVJ C00260 VJ=0.78
MOVJ C00261 VJ=0.78
MOVJ C00262 VJ=0.78
MOVL C00263 V=8.0
MOVJ C00264 VJ=0.78
MOVJ C00265 VJ=0.78
MOVJ C00266 VJ=0.78
MOVL C00267 V=8.0
MOVJ C00268 VJ=0.78
MOVJ C00269 VJ=0.78
MOVJ C00270 VJ=0.78
MOVL C00271 V=8.0
MOVJ C00272 VJ=0.78
MOVJ C00273 VJ=0.78
MOVJ C00274 VJ=0.78
MOVL C00275 V=8.0
MOVJ C00276 VJ=0.78
MOVJ C00277 VJ=0.78
MOVJ C00278 VJ=0.78
MOVL C00279 V=8.0
MOVJ C00280 VJ=0.78
MOVJ C00281 VJ=0.78
MOVJ C00282 VJ=0.78
MOVL C00283 V=8.0
MOVJ C00284 VJ=0.78
MOVJ C00285 VJ=0.78
MOVJ C00286 VJ=0.78
MOVL C00287 V=8.0
MOVJ C00288 VJ=0.78
MOVJ C00289 VJ=0.78
MOVJ C00290 VJ=0.78
MOVL C00291 V=8.0
MOVJ C00292 VJ=0.78
MOVJ C00293 VJ=0.78
MOVJ C00294 VJ=0.78
MOVL C00295 V=8.0
MOVJ C00296 VJ=0.78
MOVJ C00297 VJ=0.78
MOVJ C00298 VJ=0.78
MOVL C00299 V=8.0
MOVJ C00300 VJ=0.78
MOVJ C00301 VJ=0.78
MOVJ C00302 VJ=0.78
MOVL C00303 V=8.0
MOVJ C00304 VJ=0.78
MOVJ C00305 VJ=0.78
MOVJ C00306 VJ=0.78
MOVL C00307 V=8.0
MOVJ C00308 VJ=0.78
MOVJ C00309 VJ=0.78
MOVJ C00310 VJ=0.78
MOVL C00311 V=8.0
MOVJ C00312 VJ=0.78
MOVJ C00313 VJ=0.78
MOVJ C00314 VJ=0.78
MOVL C00315 V=8.0
MOVJ C00316 VJ=0.78
MOVJ C00317 VJ=0.78
MOVJ C00318 VJ=0.78
MOVL C00319 V=8.0
MOVJ C00320 VJ=0.78
MOVJ C00321 VJ=0.78
MOVJ C00322 VJ=0.78
MOVL C00323 V=8.0
MOVJ C00324 VJ=0.78
MOVJ C00325 VJ=0.78
MOVJ C00326 VJ=0.78
MOVL C00327 V=8.0
MOVJ C00328 VJ=0.78
MOVJ C00329 VJ=0.78
MOVJ C00330 VJ=0.78
MOVL C00331 V=8.0
MOVJ C00332 VJ=0.78
MOVJ C00333 VJ=0.78
MOVJ C00334 VJ=0.78
MOVL C00335 V=8.0
MOVJ C00336 VJ=0.78
MOVJ C00337 VJ=0.78
MOVJ C00338 VJ=0.78
MOVL C00339 V=8.0
MOVJ C00340 VJ=0.78
MOVJ C00341 VJ=0.78
MOVJ C00342 VJ=0.78
MOVL C00343 V=8.0
MOVJ C00344 VJ=0.78
MOVJ C00345 VJ=0.78
MOVJ C00346 VJ=0.78
MOVL C00347 V=8.0
MOVJ C00348 VJ=0.78
MOVJ C00349 VJ=0.78
MOVJ C00350 VJ=0.78
MOVL C00351 V=8.0
MOVJ C00352 VJ=0.78
MOVJ C00353 VJ=0.78
MOVJ C00354 VJ=0.78
MOVL C00355 V=8.0
MOVJ C00356 VJ=0.78
MOVJ C00357 VJ=0.78
MOVJ C00358 VJ=0.78
MOVL C00359 V=8.0
MOVJ C00360 VJ=0.78
MOVJ C00361 VJ=0.78
MOVJ C00362 VJ=0.78
MOVL C00363 V=8.0
MOVJ C00364 VJ=0.78
MOVJ C00365 VJ=0.78
MOVJ C00366 VJ=0.78
MOVL C00367 V=8.0
MOVJ C00368 VJ=0.78
MOVJ C00369 VJ=0.78
MOVJ C00370 VJ=0.78
MOVL C00371 V=8.0
MOVJ C00372 VJ=0.78
MOVJ C00373 VJ=0.78
MOVJ C00374 VJ=0.78
MOVL C00375 V=8.0
MOVJ C00376 VJ=0.78
MOVJ C00377 VJ=0.78
MOVJ C00378 VJ=0.78
MOVL C00379 V=8.0
MOVJ C00380 VJ=0.78
MOVJ C00381 VJ=0.78
MOVJ C00382 VJ=0.78
MOVL C00383 V=8.0
MOVJ C00384 VJ=0.78
MOVJ C00385 VJ=0.78
MOVJ C00386 VJ=0.78
MOVL C00387 V=8.0
MOVJ C00388 VJ=0.78
MOVJ C00389 VJ=0.78
MOVJ C00390 VJ=0.78
MOVL C00391 V=8.0
MOVJ C00392 VJ=0.78
MOVJ C00393 VJ=0.78
MOVJ C00394 VJ=0.78
MOVL C00395 V=8.0
MOVJ C00396 VJ=0.78
MOVJ C00397 VJ=0.78
MOVJ C00398 VJ=0.78
MOVL C00399 V=8.0
MOVJ C00400 VJ=0.78
MOVJ C00401 VJ=0.78
MOVJ C00402 VJ=0.78
MOVL C00403 V=8.0
MOVJ C00404 VJ=0.78
MOVJ C00405 VJ=0.78
MOVJ C00406 VJ=0.78
MOVL C00407 V=8.0
MOVJ C00408 VJ=0.78
MOVJ C00409 VJ=0.78
MOVJ C00410 VJ=0.78
MOVL C00411 V=8.0
MOVJ C00412 VJ=0.78
MOVJ C00413 VJ=0.78
MOVJ C00414 VJ=0.78
MOVL C00415 V=8.0
MOVJ C00416 VJ=0.78
MOVJ C00417 VJ=0.78
MOVJ C00418 VJ=0.78
MOVL C00419 V=8.0
MOVJ C00420 VJ=0.78
MOVJ C00421 VJ=0.78
MOVJ C00422 VJ=0.78
MOVL C00423 V=8.0
MOVJ C00424 VJ=0.78
MOVJ C00425 VJ=0.78
MOVJ C00426 VJ=0.78
MOVL C00427 V=8.0
MOVJ C00428 VJ=0.78
MOVJ C00429 VJ=0.78
MOVJ C00430 VJ=0.78
MOVL C00431 V=8.0
MOVJ C00432 VJ=0.78
MOVJ C00433 VJ=0.78
MOVJ C00434 VJ=0.78
MOVL C00435 V=8.0
MOVJ C00436 VJ=0.78
MOVJ C00437 VJ=0.78
MOVJ C00438 VJ=0.78
MOVL C00439 V=8.0
MOVJ C00440 VJ=0.78
MOVJ C00441 VJ=0.78
MOVJ C00442 VJ=0.78
MOVL C00443 V=8.0
MOVJ C00444 VJ=0.78
MOVJ C00445 VJ=0.78
MOVJ C00446 VJ=0.78
MOVL C00447 V=8.0
MOVJ C00448 VJ=0.78
MOVJ C00449 VJ=0.78
MOVJ C00450 VJ=0.78
MOVL C00451 V=8.0
MOVJ C00452 VJ=0.78
MOVJ C00453 VJ=0.78
MOVJ C00454 VJ=0.78
MOVL C00455 V=8.0
MOVJ C00456 VJ=0.78
MOVJ C00457 VJ=0.78
MOVJ C00458 VJ=0.78
MOVL C00459 V=8.0
MOVJ C00460 VJ=0.78
MOVJ C00461 VJ=0.78
MOVJ C00462 VJ=0.78
MOVL C00463 V=8.0
MOVJ C00464 VJ=0.78
MOVJ C00465 VJ=0.78
MOVJ C00466 VJ=0.78
MOVL C00467 V=8.0
MOVJ C00468 VJ=0.78
MOVJ C00469 VJ=0.78
MOVJ C00470 VJ=0.78
MOVL C00471 V=8.0
MOVJ C00472 VJ=0.78
MOVJ C00473 VJ=0.78
MOVJ C00474 VJ=0.78
MOVL C00475 V=8.0
MOVJ C00476 VJ=0.78
MOVJ C00477 VJ=0.78
MOVJ C00478 VJ=0.78
MOVL C00479 V=8.0
MOVJ C00480 VJ=0.78
MOVJ C00481 VJ=0.78
MOVJ C00482 VJ=0.78
MOVL C00483 V=8.0
MOVJ C00484 VJ=0.78
MOVJ C00485 VJ=0.78
MOVJ C00486 VJ=0.78
MOVL C00487 V=8.0
MOVJ C00488 VJ=0.78
MOVJ C00489 VJ=0.78
MOVJ C00490 VJ=0.78
MOVL C00491 V=8.0
MOVJ C00492 VJ=0.78
MOVJ C00493 VJ=0.78
MOVJ C00494 VJ=0.78
MOVL C00495 V=8.0
MOVJ C00496 VJ=0.78
MOVJ C00497 VJ=0.78
MOVJ C00498 VJ=0.78
MOVL C00499 V=8.0
MOVJ C00500 VJ=0.78
MOVJ C00501 VJ=0.78
MOVJ C00502 VJ=0.78
MOVL C00503 V=8.0
MOVJ C00504 VJ=0.78
MOVJ C00505 VJ=0.78
MOVJ C00506 VJ=0.78
MOVL C00507 V=8.0
MOVJ C00508 VJ=0.78
MOVJ C00509 VJ=0.78
MOVJ C00510 VJ=0.78
MOVL C00511 V=8.0
MOVJ C00512 VJ=0.78
MOVJ C00513 VJ=0.78
MOVJ C00514 VJ=0.78
MOVL C00515 V=8.0
MOVJ C00516 VJ=0.78
MOVJ C00517 VJ=0.78
MOVJ C00518 VJ=0.78
MOVL C00519 V=8.0
MOVJ C00520 VJ=0.78
MOVJ C00521 VJ=0.78
MOVJ C00522 VJ=0.78
MOVL C00523 V=8.0
MOVJ C00524 VJ=0.78
MOVJ C00525 VJ=0.78
MOVJ C00526 VJ=0.78
MOVL C00527 V=8.0
MOVJ C00528 VJ=0.78
MOVJ C00529 VJ=0.78
MOVJ C00530 VJ=0.78
MOVL C00531 V=8.0
MOVJ C00532 VJ=0.78
MOVJ C00533 VJ=0.78
MOVJ C00534 VJ=0.78
MOVL C00535 V=8.0
MOVJ C00536 VJ=0.78
MOVJ C00537 VJ=0.78
MOVJ C00538 VJ=0.78
MOVL C00539 V=8.0
MOVJ C00540 VJ=0.78
MOVJ C00541 VJ=0.78
MOVJ C00542 VJ=0.78
MOVL C00543 V=8.0
MOVJ C00544 VJ=0.78
MOVJ C00545 VJ=0.78
MOVJ C00546 VJ=0.78
MOVL C00547 V=8.0
MOVJ C00548 VJ=0.78
MOVJ C00549 VJ=0.78
MOVJ C00550 VJ=0.78
MOVL C00551 V=8.0
MOVJ C00552 VJ=0.78
MOVJ C00553 VJ=0.78
MOVJ C00554 VJ=0.78
MOVL C00555 V=8.0
MOVJ C00556 VJ=0.78
MOVJ C00557 VJ=0.78
MOVJ C00558 VJ=0.78
MOVL C00559 V=8.0
MOVJ C00560 VJ=0.78
MOVJ C00561 VJ=0.78
MOVJ C00562 VJ=0.78
MOVL C00563 V=8.0
MOVJ C00564 VJ=0.78
MOVJ C00565 VJ=0.78
MOVJ C00566 VJ=0.78
MOVL C00567 V=8.0
MOVJ C00568 VJ=0.78
MOVJ C00569 VJ=0.78
MOVJ C00570 VJ=0.78
MOVL C00571 V=8.0
MOVJ C00572 VJ=0.78
MOVJ C00573 VJ=0.78
MOVJ C00574 VJ=0.78
MOVL C00575 V=8.0
MOVJ C00576 VJ=0.78
MOVJ C00577 VJ=0.78
MOVJ C00578 VJ=0.78
MOVL C00579 V=8.0
MOVJ C00580 VJ=0.78
MOVJ C00581 VJ=0.78
MOVJ C00582 VJ=0.78
MOVL C00583 V=8.0
MOVJ C00584 VJ=0.78
MOVJ C00585 VJ=0.78
MOVJ C00586 VJ=0.78
MOVL C00587 V=8.0
MOVJ C00588 VJ=0.78
MOVJ C00589 VJ=0.78
MOVJ C00590 VJ=0.78
MOVL C00591 V=8.0
MOVJ C00592 VJ=0.78
MOVJ C00593 VJ=0.78
MOVJ C00594 VJ=0.78
MOVL C00595 V=8.0
MOVJ C00596 VJ=0.78
MOVJ C00597 VJ=0.78
MOVJ C00598 VJ=0.78
MOVL C00599 V=8.0
MOVJ C00600 VJ=0.78
MOVJ C00601 VJ=0.78
MOVJ C00602 VJ=0.78
MOVL C00603 V=8.0
MOVJ C00604 VJ=0.78
MOVJ C00605 VJ=0.78
MOVJ C00606 VJ=0.78
MOVL C00607 V=8.0
MOVJ C00608 VJ=0.78
MOVJ C00609 VJ=0.78
MOVJ C00610 VJ=0.78
MOVL C00611 V=8.0
MOVJ C00612 VJ=0.78
MOVJ C00613 VJ=0.78
MOVJ C00614 VJ=0.78
MOVL C00615 V=8.0
MOVJ C00616 VJ=0.78
MOVJ C00617 VJ=0.78
MOVJ C00618 VJ=0.78
MOVL C00619 V=8.0
MOVJ C00620 VJ=0.78
MOVJ C00621 VJ=0.78
MOVJ C00622 VJ=0.78
MOVL C00623 V=8.0
MOVJ C00624 VJ=0.78
MOVJ C00625 VJ=0.78
MOVJ C00626 VJ=0.78
MOVL C00627 V=8.0
MOVJ C00628 VJ=0.78
MOVJ C00629 VJ=0.78
MOVJ C00630 VJ=0.78
MOVL C00631 V=8.0
MOVJ C00632 VJ=0.78
MOVJ C00633 VJ=0.78
MOVJ C00634 VJ=0.78
MOVL C00635 V=8.0
MOVJ C00636 VJ=0.78
MOVJ C00637 VJ=0.78
MOVJ C00638 VJ=0.78
MOVL C00639 V=8.0
MOVJ C00640 VJ=0.78
MOVJ C00641 VJ=0.78
MOVJ C00642 VJ=0.78
MOVL C00643 V=8.0
MOVJ C00644 VJ=0.78
MOVJ C00645 VJ=0.78
MOVJ C00646 VJ=0.78
MOVL C00647 V=8.0
MOVJ C00648 VJ=0.78
MOVJ C00649 VJ=0.78
MOVJ C00650 VJ=0.78
MOVL C00651 V=8.0
MOVJ C00652 VJ=0.78
MOVJ C00653 VJ=0.78
MOVJ C00654 VJ=0.78
MOVL C00655 V=8.0
MOVJ C00656 VJ=0.78
MOVJ C00657 VJ=0.78
MOVJ C00658 VJ=0.78
MOVL C00659 V=8.0
MOVJ C00660 VJ=0.78
MOVJ C00661 VJ=0.78
MOVJ C00662 VJ=0.78
MOVL C00663 V=8.0
MOVJ C00664 VJ=0.78
MOVJ C00665 VJ=0.78
MOVJ C00666 VJ=0.78
MOVL C00667 V=8.0
MOVJ C00668 VJ=0.78
MOVJ C00669 VJ=0.78
MOVJ C00670 VJ=0.78
MOVL C00671 V=8.0
MOVJ C00672 VJ=0.78
MOVJ C00673 VJ=0.78
MOVJ C00674 VJ=0.78
MOVL C00675 V=8.0
MOVJ C00676 VJ=0.78
MOVJ C00677 VJ=0.78
MOVJ C00678 VJ=0.78
MOVL C00679 V=8.0
MOVJ C00680 VJ=0.78
MOVJ C00681 VJ=0.78
MOVJ C00682 VJ=0.78
MOVL C00683 V=8.0
MOVJ C00684 VJ=0.78
MOVJ C00685 VJ=0.78
MOVJ C00686 VJ=0.78
MOVL C00687 V=8.0
MOVJ C00688 VJ=0.78
MOVJ C00689 VJ=0.78
MOVJ C00690 VJ=0.78
MOVL C00691 V=8.0
MOVJ C00692 VJ=0.78
MOVJ C00693 VJ=0.78
MOVJ C00694 VJ=0.78
MOVL C00695 V=8.0
MOVJ C00696 VJ=0.78
MOVJ C00697 VJ=0.78
MOVJ C00698 VJ=0.78
MOVL C00699 V=8.0
MOVJ C00700 VJ=0.78
MOVJ C00701 VJ=0.78
MOVJ C00702 VJ=0.78
MOVL C00703 V=8.0
MOVJ C00704 VJ=0.78
MOVJ C00705 VJ=0.78
MOVJ C00706 VJ=0.78
MOVL C00707 V=8.0
MOVJ C00708 VJ=0.78
MOVJ C00709 VJ=0.78
MOVJ C00710 VJ=0.78
MOVL C00711 V=8.0
MOVJ C00712 VJ=0.78
MOVJ C00713 VJ=0.78
MOVJ C00714 VJ=0.78
MOVL C00715 V=8.0
MOVJ C00716 VJ=0.78
MOVJ C00717 VJ=0.78
MOVJ C00718 VJ=0.78
MOVL C00719 V=8.0
MOVJ C00720 VJ=0.78
MOVJ C00721 VJ=0.78
MOVJ C00722 VJ=0.78
MOVL C00723 V=8.0
MOVJ C00724 VJ=0.78
MOVJ C00725 VJ=0.78
MOVJ C00726 VJ=0.78
MOVL C00727 V=8.0
MOVJ C00728 VJ=0.78
MOVJ C00729 VJ=0.78
MOVJ C00730 VJ=0.78
MOVL C00731 V=8.0
MOVJ C00732 VJ=0.78
MOVJ C00733 VJ=0.78
MOVJ C00734 VJ=0.78
MOVL C00735 V=8.0
MOVJ C00736 VJ=0.78
MOVJ C00737 VJ=0.78
MOVJ C00738 VJ=0.78
MOVL C00739 V=8.0
MOVJ C00740 VJ=0.78
MOVJ C00741 VJ=0.78
MOVJ C00742 VJ=0.78
MOVL C00743 V=8.0
MOVJ C00744 VJ=0.78
MOVJ C00745 VJ=0.78
MOVJ C00746 VJ=0.78
MOVL C00747 V=8.0
MOVJ C00748 VJ=0.78
MOVJ C00749 VJ=0.78
MOVJ C00750 VJ=0.78
MOVL C00751 V=8.0
MOVJ C00752 VJ=0.78
MOVJ C00753 VJ=0.78
MOVJ C00754 VJ=0.78
MOVL C00755 V=8.0
MOVJ C00756 VJ=0.78
MOVJ C00757 VJ=0.78
MOVJ C00758 VJ=0.78
MOVL C00759 V=8.0
MOVJ C00760 VJ=0.78
MOVJ C00761 VJ=0.78
MOVJ C00762 VJ=0.78
MOVL C00763 V=8.0
MOVJ C00764 VJ=0.78
MOVJ C00765 VJ=0.78
MOVJ C00766 VJ=0.78
MOVL C00767 V=8.0
MOVJ C00768 VJ=0.78
MOVJ C00769 VJ=0.78
MOVJ C00770 VJ=0.78
MOVL C00771 V=8.0
MOVJ C00772 VJ=0.78
MOVJ C00773 VJ=0.78
MOVJ C00774 VJ=0.78
MOVL C00775 V=8.0
MOVJ C00776 VJ=0.78
MOVJ C00777 VJ=0.78
MOVJ C00778 VJ=0.78
MOVL C00779 V=8.0
MOVJ C00780 VJ=0.78
MOVJ C00781 VJ=0.78
MOVJ C00782 VJ=0.78
MOVL C00783 V=8.0
MOVJ C00784 VJ=0.78
MOVJ C00785 VJ=0.78
MOVJ C00786 VJ=0.78
MOVL C00787 V=8.0
MOVJ C00788 VJ=0.78
MOVJ C00789 VJ=0.78
MOVJ C00790 VJ=0.78
MOVL C00791 V=8.0
MOVJ C00792 VJ=0.78
MOVJ C00793 VJ=0.78
MOVJ C00794 VJ=0.78
MOVL C00795 V=8.0
MOVJ C00796 VJ=0.78
MOVJ C00797 VJ=0.78
MOVJ C00798 VJ=0.78
MOVL C00799 V=8.0
MOVJ C00800 VJ=0.78
MOVJ C00801 VJ=0.78
MOVJ C00802 VJ=0.78
MOVL C00803 V=8.0
MOVJ C00804 VJ=0.78
MOVJ C00805 VJ=0.78
MOVJ C00806 VJ=0.78
MOVL C00807 V=8.0
MOVJ C00808 VJ=0.78
MOVJ C00809 VJ=0.78
MOVJ C00810 VJ=0.78
MOVL C00811 V=8.0
MOVJ C00812 VJ=0.78
MOVJ C00813 VJ=0.78
MOVJ C00814 VJ=0.78
MOVL C00815 V=8.0
MOVJ C00816 VJ=0.78
MOVJ C00817 VJ=0.78
MOVJ C00818 VJ=0.78
MOVL C00819 V=8.0
MOVJ C00820 VJ=0.78
MOVJ C00821 VJ=0.78
MOVJ C00822 VJ=0.78
MOVL C00823 V=8.0
MOVJ C00824 VJ=0.78
MOVJ C00825 VJ=0.78
MOVJ C00826 VJ=0.78
MOVL C00827 V=8.0
MOVJ C00828 VJ=0.78
MOVJ C00829 VJ=0.78
MOVJ C00830 VJ=0.78
MOVL C00831 V=8.0
MOVJ C00832 VJ=0.78
MOVJ C00833 VJ=0.78
MOVJ C00834 VJ=0.78
MOVL C00835 V=8.0
MOVJ C00836 VJ=0.78
MOVJ C00837 VJ=0.78
MOVJ C00838 VJ=0.78
MOVL C00839 V=8.0
MOVJ C00840 VJ=0.78
MOVJ C00841 VJ=0.78
MOVJ C00842 VJ=0.78
MOVL C00843 V=8.0
MOVJ C00844 VJ=0.78
MOVJ C00845 VJ=0.78
MOVJ C00846 VJ=0.78
MOVL C00847 V=8.0
MOVJ C00848 VJ=0.78
MOVJ C00849 VJ=0.78
MOVJ C00850 VJ=0.78
MOVL C00851 V=8.0
MOVJ C00852 VJ=0.78
MOVJ C00853 VJ=0.78
MOVJ C00854 VJ=0.78
MOVL C00855 V=8.0
MOVJ C00856 VJ=0.78
MOVJ C00857 VJ=0.78
MOVJ C00858 VJ=0.78
MOVL C00859 V=8.0
MOVJ C00860 VJ=0.78
MOVJ C00861 VJ=0.78
MOVJ C00862 VJ=0.78
MOVL C00863 V=8.0
MOVJ C00864 VJ=0.78
MOVJ C00865 VJ=0.78
MOVJ C00866 VJ=0.78
MOVL C00867 V=8.0
MOVJ C00868 VJ=0.78
MOVJ C00869 VJ=0.78
MOVJ C00870 VJ=0.78
MOVL C00871 V=8.0
MOVJ C00872 VJ=0.78
MOVJ C00873 VJ=0.78
MOVJ C00874 VJ=0.78
MOVL C00875 V=8.0
MOVJ C00876 VJ=0.78
MOVJ C00877 VJ=0.78
MOVJ C00878 VJ=0.78
MOVL C00879 V=8.0
MOVJ C00880 VJ=0.78
MOVJ C00881 VJ=0.78
MOVJ C00882 VJ=0.78
MOVL C00883 V=8.0
MOVJ C00884 VJ=0.78
MOVJ C00885 VJ=0.78
MOVJ C00886 VJ=0.78
MOVL C00887 V=8.0
MOVJ C00888 VJ=0.78
MOVJ C00889 VJ=0.78
MOVJ C00890 VJ=0.78
MOVL C00891 V=8.0
MOVJ C00892 VJ=0.78
MOVJ C00893 VJ=0.78
MOVJ C00894 VJ=0.78
MOVL C00895 V=8.0
MOVJ C00896 VJ=0.78
MOVJ C00897 VJ=0.78
MOVJ C00898 VJ=0.78
MOVL C00899 V=8.0
MOVJ C00900 VJ=0.78
MOVJ C00901 VJ=0.78
MOVJ C00902 VJ=0.78
MOVL C00903 V=8.0
MOVJ C00904 VJ=0.78
MOVJ C00905 VJ=0.78
MOVJ C00906 VJ=0.78
MOVL C00907 V=8.0
MOVJ C00908 VJ=0.78
MOVJ C00909 VJ=0.78
MOVJ C00910 VJ=0.78
MOVL C00911 V=8.0
MOVJ C00912 VJ=0.78
MOVJ C00913 VJ=0.78
MOVJ C00914 VJ=0.78
MOVL C00915 V=8.0
MOVJ C00916 VJ=0.78
MOVJ C00917 VJ=0.78
MOVJ C00918 VJ=0.78
MOVL C00919 V=8.0
MOVJ C00920 VJ=0.78
MOVJ C00921 VJ=0.78
MOVJ C00922 VJ=0.78
MOVL C00923 V=8.0
MOVJ C00924 VJ=0.78
MOVJ C00925 VJ=0.78
MOVJ C00926 VJ=0.78
MOVL C00927 V=8.0
MOVJ C00928 VJ=0.78
MOVJ C00929 VJ=0.78
MOVJ C00930 VJ=0.78
MOVL C00931 V=8.0
MOVJ C00932 VJ=0.78
MOVJ C00933 VJ=0.78
MOVJ C00934 VJ=0.78
MOVL C00935 V=8.0
MOVJ C00936 VJ=0.78
MOVJ C00937 VJ=0.78
MOVJ C00938 VJ=0.78
MOVL C00939 V=8.0
MOVJ C00940 VJ=0.78
MOVJ C00941 VJ=0.78
MOVJ C00942 VJ=0.78
MOVL C00943 V=8.0
MOVJ C00944 VJ=0.78
MOVJ C00945 VJ=0.78
MOVJ C00946 VJ=0.78
MOVL C00947 V=8.0
MOVJ C00948 VJ=0.78
MOVJ C00949 VJ=0.78
MOVJ C00950 VJ=0.78
MOVL C00951 V=8.0
MOVJ C00952 VJ=0.78
MOVJ C00953 VJ=0.78
MOVJ C00954 VJ=0.78
MOVL C00955 V=8.0
MOVJ C00956 VJ=0.78
MOVJ C00957 VJ=0.78
MOVJ C00958 VJ=0.78
MOVL C00959 V=8.0
MOVJ C00960 VJ=0.78
MOVJ C00961 VJ=0.78
MOVJ C00962 VJ=0.78
MOVL C00963 V=8.0
MOVJ C00964 VJ=0.78
MOVJ C00965 VJ=0.78
MOVJ C00966 VJ=0.78
MOVL C00967 V=8.0
MOVJ C00968 VJ=0.78
MOVJ C00969 VJ=0.78
MOVJ C00970 VJ=0.78
MOVL C00971 V=8.0
MOVJ C00972 VJ=0.78
MOVJ C00973 VJ=0.78
MOVJ C00974 VJ=0.78
MOVL C00975 V=8.0
MOVJ C00976 VJ=0.78
MOVJ C00977 VJ=0.78
MOVJ C00978 VJ=0.78
MOVL C00979 V=8.0
MOVJ C00980 VJ=0.78
MOVJ C00981 VJ=0.78
MOVJ C00982 VJ=0.78
MOVL C00983 V=8.0
MOVJ C00984 VJ=0.78
MOVJ C00985 VJ=0.78
MOVJ C00986 VJ=0.78
MOVL C00987 V=8.0
MOVJ C00988 VJ=0.78
MOVJ C00989 VJ=0.78
MOVJ C00990 VJ=0.78
MOVL C00991 V=8.0
MOVJ C00992 VJ=0.78
MOVJ C00993 VJ=0.78
MOVJ C00994 VJ=0.78
MOVL C00995 V=8.0
MOVJ C00996 VJ=0.78
MOVJ C00997 VJ=0.78
MOVJ C00998 VJ=0.78
MOVL C00999 V=8.0
MOVJ C01000 VJ=0.78
MOVJ C01001 VJ=0.78
MOVJ C01002 VJ=0.78
MOVL C01003 V=8.0
MOVJ C01004 VJ=0.78
MOVJ C01005 VJ=0.78
MOVJ C01006 VJ=0.78
MOVL C01007 V=8.0
MOVJ C01008 VJ=0.78
MOVJ C01009 VJ=0.78
MOVJ C01010 VJ=0.78
MOVL C01011 V=8.0
MOVJ C01012 VJ=0.78
MOVJ C01013 VJ=0.78
MOVJ C01014 VJ=0.78
MOVL C01015 V=8.0
MOVJ C01016 VJ=0.78
MOVJ C01017 VJ=0.78
MOVJ C01018 VJ=0.78
MOVL C01019 V=8.0
MOVJ C01020 VJ=0.78
MOVJ C01021 VJ=0.78
MOVJ C01022 VJ=0.78
MOVL C01023 V=8.0
MOVJ C01024 VJ=0.78
MOVJ C01025 VJ=0.78
MOVJ C01026 VJ=0.78
MOVL C01027 V=8.0
MOVJ C01028 VJ=0.78
MOVJ C01029 VJ=0.78
MOVJ C01030 VJ=0.78
MOVL C01031 V=8.0
MOVJ C01032 VJ=0.78
MOVJ C01033 VJ=0.78
MOVJ C01034 VJ=0.78
MOVL C01035 V=8.0
MOVJ C01036 VJ=0.78
MOVJ C01037 VJ=0.78
MOVJ C01038 VJ=0.78
MOVL C01039 V=8.0
MOVJ C01040 VJ=0.78
MOVJ C01041 VJ=0.78
MOVJ C01042 VJ=0.78
MOVL C01043 V=8.0
MOVJ C01044 VJ=0.78
MOVJ C01045 VJ=0.78
MOVJ C01046 VJ=0.78
MOVL C01047 V=8.0
MOVJ C01048 VJ=0.78
MOVJ C01049 VJ=0.78
MOVJ C01050 VJ=0.78
MOVL C01051 V=8.0
MOVJ C01052 VJ=0.78
MOVJ C01053 VJ=0.78
MOVJ C01054 VJ=0.78
MOVL C01055 V=8.0
MOVJ C01056 VJ=0.78
MOVJ C01057 VJ=0.78
MOVJ C01058 VJ=0.78
MOVL C01059 V=8.0
MOVJ C01060 VJ=0.78
MOVJ C01061 VJ=0.78
MOVJ C01062 VJ=0.78
MOVL C01063 V=8.0
MOVJ C01064 VJ=0.78
MOVJ C01065 VJ=0.78
MOVJ C01066 VJ=0.78
MOVL C01067 V=8.0
MOVJ C01068 VJ=0.78
MOVJ C01069 VJ=0.78
MOVJ C01070 VJ=0.78
MOVL C01071 V=8.0
MOVJ C01072 VJ=0.78
MOVJ C01073 VJ=0.78
MOVJ C01074 VJ=0.78
MOVL C01075 V=8.0
MOVJ C01076 VJ=0.78
MOVJ C01077 VJ=0.78
MOVJ C01078 VJ=0.78
MOVL C01079 V=8.0
MOVJ C01080 VJ=0.78
MOVJ C01081 VJ=0.78
MOVJ C01082 VJ=0.78
MOVL C01083 V=8.0
MOVJ C01084 VJ=0.78
MOVJ C01085 VJ=0.78
MOVJ C01086 VJ=0.78
MOVL C01087 V=8.0
MOVJ C01088 VJ=0.78
MOVJ C01089 VJ=0.78
MOVJ C01090 VJ=0.78
MOVL C01091 V=8.0
MOVJ C01092 VJ=0.78
MOVJ C01093 VJ=0.78
MOVJ C01094 VJ=0.78
MOVL C01095 V=8.0
MOVJ C01096 VJ=0.78
MOVJ C01097 VJ=0.78
MOVJ C01098 VJ=0.78
MOVL C01099 V=8.0
MOVJ C01100 VJ=0.78
MOVJ C01101 VJ=0.78
MOVJ C01102 VJ=0.78
MOVL C01103 V=8.0
MOVJ C01104 VJ=0.78
MOVJ C01105 VJ=0.78
MOVJ C01106 VJ=0.78
MOVL C01107 V=8.0
MOVJ C01108 VJ=0.78
MOVJ C01109 VJ=0.78
MOVJ C01110 VJ=0.78
MOVL C01111 V=8.0
MOVJ C01112 VJ=0.78
MOVJ C01113 VJ=0.78
MOVJ C01114 VJ=0.78
MOVL C01115 V=8.0
MOVJ C01116 VJ=0.78
MOVJ C01117 VJ=0.78
MOVJ C01118 VJ=0.78
MOVL C01119 V=8.0
MOVJ C01120 VJ=0.78
MOVJ C01121 VJ=0.78
MOVJ C01122 VJ=0.78
MOVL C01123 V=8.0
MOVJ C01124 VJ=0.78
MOVJ C01125 VJ=0.78
MOVJ C01126 VJ=0.78
MOVL C01127 V=8.0
MOVJ C01128 VJ=0.78
MOVJ C01129 VJ=0.78
MOVJ C01130 VJ=0.78
MOVL C01131 V=8.0
MOVJ C01132 VJ=0.78
MOVJ C01133 VJ=0.78
MOVJ C01134 VJ=0.78
MOVL C01135 V=8.0
MOVJ C01136 VJ=0.78
MOVJ C01137 VJ=0.78
MOVJ C01138 VJ=0.78
MOVL C01139 V=8.0
MOVJ C01140 VJ=0.78
MOVJ C01141 VJ=0.78
MOVJ C01142 VJ=0.78
MOVL C01143 V=8.0
MOVJ C01144 VJ=0.78
MOVJ C01145 VJ=0.78
MOVJ C01146 VJ=0.78
MOVL C01147 V=8.0
MOVJ C01148 VJ=0.78
MOVJ C01149 VJ=0.78
MOVJ C01150 VJ=0.78
MOVL C01151 V=8.0
MOVJ C01152 VJ=0.78
MOVJ C01153 VJ=0.78
MOVJ C01154 VJ=0.78
MOVL C01155 V=8.0
MOVJ C01156 VJ=0.78
MOVJ C01157 VJ=0.78
MOVJ C01158 VJ=0.78
MOVL C01159 V=8.0
MOVJ C01160 VJ=0.78
MOVJ C01161 VJ=0.78
MOVJ C01162 VJ=0.78
MOVL C01163 V=8.0
MOVJ C01164 VJ=0.78
MOVJ C01165 VJ=0.78
MOVJ C01166 VJ=0.78
MOVL C01167 V=8.0
MOVJ C01168 VJ=0.78
MOVJ C01169 VJ=0.78
MOVJ C01170 VJ=0.78
MOVL C01171 V=8.0
MOVJ C01172 VJ=0.78
MOVJ C01173 VJ=0.78
MOVJ C01174 VJ=0.78
MOVL C01175 V=8.0
MOVJ C01176 VJ=0.78
MOVJ C01177 VJ=0.78
MOVJ C01178 VJ=0.78
MOVL C01179 V=8.0
MOVJ C01180 VJ=0.78
MOVJ C01181 VJ=0.78
MOVJ C01182 VJ=0.78
MOVL C01183 V=8.0
MOVJ C01184 VJ=0.78
MOVJ C01185 VJ=0.78
MOVJ C01186 VJ=0.78
MOVL C01187 V=8.0
MOVJ C01188 VJ=0.78
MOVJ C01189 VJ=0.78
MOVJ C01190 VJ=0.78
MOVL C01191 V=8.0
MOVJ C01192 VJ=0.78
MOVJ C01193 VJ=0.78
MOVJ C01194 VJ=0.78
MOVL C01195 V=8.0
MOVJ C01196 VJ=0.78
MOVJ C01197 VJ=0.78
MOVJ C01198 VJ=0.78
MOVL C01199 V=8.0
MOVJ C01200 VJ=0.78
MOVJ C01201 VJ=0.78
MOVJ C01202 VJ=0.78
MOVL C01203 V=8.0
MOVJ C01204 VJ=0.78
MOVJ C01205 VJ=0.78
MOVJ C01206 VJ=0.78
MOVL C01207 V=8.0
MOVJ C01208 VJ=0.78
MOVJ C01209 VJ=0.78
MOVJ C01210 VJ=0.78
MOVL C01211 V=8.0
MOVJ C01212 VJ=0.78
MOVJ C01213 VJ=0.78
MOVJ C01214 VJ=0.78
MOVL C01215 V=8.0
MOVJ C01216 VJ=0.78
MOVJ C01217 VJ=0.78
MOVJ C01218 VJ=0.78
MOVL C01219 V=8.0
MOVJ C01220 VJ=0.78
MOVJ C01221 VJ=0.78
MOVJ C01222 VJ=0.78
MOVL C01223 V=8.0
MOVJ C01224 VJ=0.78
MOVJ C01225 VJ=0.78
MOVJ C01226 VJ=0.78
MOVL C01227 V=8.0
MOVJ C01228 VJ=0.78
MOVJ C01229 VJ=0.78
MOVJ C01230 VJ=0.78
MOVL C01231 V=8.0
MOVJ C01232 VJ=0.78
MOVJ C01233 VJ=0.78
MOVJ C01234 VJ=0.78
MOVL C01235 V=8.0
MOVJ C01236 VJ=0.78
MOVJ C01237 VJ=0.78
MOVJ C01238 VJ=0.78
MOVL C01239 V=8.0
MOVJ C01240 VJ=0.78
MOVJ C01241 VJ=0.78
MOVJ C01242 VJ=0.78
MOVL C01243 V=8.0
MOVJ C01244 VJ=0.78
MOVJ C01245 VJ=0.78
MOVJ C01246 VJ=0.78
MOVL C01247 V=8.0
MOVJ C01248 VJ=0.78
MOVJ C01249 VJ=0.78
MOVJ C01250 VJ=0.78
MOVL C01251 V=8.0
MOVJ C01252 VJ=0.78
MOVJ C01253 VJ=0.78
MOVJ C01254 VJ=0.78
MOVL C01255 V=8.0
MOVJ C01256 VJ=0.78
MOVJ C01257 VJ=0.78
MOVJ C01258 VJ=0.78
MOVL C01259 V=8.0
MOVJ C01260 VJ=0.78
MOVJ C01261 VJ=0.78
MOVJ C01262 VJ=0.78
MOVL C01263 V=8.0
MOVJ C01264 VJ=0.78
MOVJ C01265 VJ=0.78
MOVJ C01266 VJ=0.78
MOVL C01267 V=8.0
MOVJ C01268 VJ=0.78
MOVJ C01269 VJ=0.78
MOVJ C01270 VJ=0.78
MOVL C01271 V=8.0
MOVJ C01272 VJ=0.78
MOVJ C01273 VJ=0.78
MOVJ C01274 VJ=0.78
MOVL C01275 V=8.0
MOVJ C01276 VJ=0.78
MOVJ C01277 VJ=0.78
MOVJ C01278 VJ=0.78
MOVL C01279 V=8.0
MOVJ C01280 VJ=0.78
MOVJ C01281 VJ=0.78
MOVJ C01282 VJ=0.78
MOVL C01283 V=8.0
MOVJ C01284 VJ=0.78
MOVJ C01285 VJ=0.78
MOVJ C01286 VJ=0.78
MOVL C01287 V=8.0
MOVJ C01288 VJ=0.78
MOVJ C01289 VJ=0.78
MOVJ C01290 VJ=0.78
MOVL C01291 V=8.0
MOVJ C01292 VJ=0.78
MOVJ C01293 VJ=0.78
MOVJ C01294 VJ=0.78
MOVL C01295 V=8.0
MOVJ C01296 VJ=0.78
MOVJ C01297 VJ=0.78
MOVJ C01298 VJ=0.78
MOVL C01299 V=8.0
MOVJ C01300 VJ=0.78
MOVJ C01301 VJ=0.78
MOVJ C01302 VJ=0.78
MOVL C01303 V=8.0
MOVJ C01304 VJ=0.78
MOVJ C01305 VJ=0.78
MOVJ C01306 VJ=0.78
MOVL C01307 V=8.0
MOVJ C01308 VJ=0.78
MOVJ C01309 VJ=0.78
MOVJ C01310 VJ=0.78
MOVL C01311 V=8.0
MOVJ C01312 VJ=0.78
MOVJ C01313 VJ=0.78
MOVJ C01314 VJ=0.78
MOVL C01315 V=8.0
MOVJ C01316 VJ=0.78
MOVJ C01317 VJ=0.78
MOVJ C01318 VJ=0.78
MOVL C01319 V=8.0
MOVJ C01320 VJ=0.78
MOVJ C01321 VJ=0.78
MOVJ C01322 VJ=0.78
MOVL C01323 V=8.0
MOVJ C01324 VJ=0.78
MOVJ C01325 VJ=0.78
MOVJ C01326 VJ=0.78
MOVL C01327 V=8.0
MOVJ C01328 VJ=0.78
MOVJ C01329 VJ=0.78
MOVJ C01330 VJ=0.78
MOVL C01331 V=8.0
MOVJ C01332 VJ=0.78
MOVJ C01333 VJ=0.78
MOVJ C01334 VJ=0.78
MOVL C01335 V=8.0
MOVJ C01336 VJ=0.78
MOVJ C01337 VJ=0.78
MOVJ C01338 VJ=0.78
MOVL C01339 V=8.0
MOVJ C01340 VJ=0.78
MOVJ C01341 VJ=0.78
MOVJ C01342 VJ=0.78
MOVL C01343 V=8.0
MOVJ C01344 VJ=0.78
MOVJ C01345 VJ=0.78
MOVJ C01346 VJ=0.78
MOVL C01347 V=8.0
MOVJ C01348 VJ=0.78
MOVJ C01349 VJ=0.78
MOVJ C01350 VJ=0.78
MOVL C01351 V=8.0
MOVJ C01352 VJ=0.78
MOVJ C01353 VJ=0.78
MOVJ C01354 VJ=0.78
MOVL C01355 V=8.0
MOVJ C01356 VJ=0.78
MOVJ C01357 VJ=0.78
MOVJ C01358 VJ=0.78
MOVL C01359 V=8.0
MOVJ C01360 VJ=0.78
MOVJ C01361 VJ=0.78
MOVJ C01362 VJ=0.78
MOVL C01363 V=8.0
MOVJ C01364 VJ=0.78
MOVJ C01365 VJ=0.78
MOVJ C01366 VJ=0.78
MOVL C01367 V=8.0
MOVJ C01368 VJ=0.78
MOVJ C01369 VJ=0.78
MOVJ C01370 VJ=0.78
MOVL C01371 V=8.0
MOVJ C01372 VJ=0.78
MOVJ C01373 VJ=0.78
MOVJ C01374 VJ=0.78
MOVL C01375 V=8.0
MOVJ C01376 VJ=0.78
MOVJ C01377 VJ=0.78
MOVJ C01378 VJ=0.78
MOVL C01379 V=8.0
MOVJ C01380 VJ=0.78
MOVJ C01381 VJ=0.78
MOVJ C01382 VJ=0.78
MOVL C01383 V=8.0
MOVJ C01384 VJ=0.78
MOVJ C01385 VJ=0.78
MOVJ C01386 VJ=0.78
MOVL C01387 V=8.0
MOVJ C01388 VJ=0.78
MOVJ C01389 VJ=0.78
MOVJ C01390 VJ=0.78
MOVL C01391 V=8.0
MOVJ C01392 VJ=0.78
MOVJ C01393 VJ=0.78
MOVJ C01394 VJ=0.78
MOVL C01395 V=8.0
MOVJ C01396 VJ=0.78
MOVJ C01397 VJ=0.78
MOVJ C01398 VJ=0.78
MOVL C01399 V=8.0
MOVJ C01400 VJ=0.78
MOVJ C01401 VJ=0.78
MOVJ C01402 VJ=0.78
MOVL C01403 V=8.0
MOVJ C01404 VJ=0.78
MOVJ C01405 VJ=0.78
MOVJ C01406 VJ=0.78
MOVL C01407 V=8.0
MOVJ C01408 VJ=0.78
MOVJ C01409 VJ=0.78
MOVJ C01410 VJ=0.78
MOVL C01411 V=8.0
MOVJ C01412 VJ=0.78
MOVJ C01413 VJ=0.78
MOVJ C01414 VJ=0.78
MOVL C01415 V=8.0
MOVJ C01416 VJ=0.78
MOVJ C01417 VJ=0.78
MOVJ C01418 VJ=0.78
MOVL C01419 V=8.0
MOVJ C01420 VJ=0.78
MOVJ C01421 VJ=0.78
MOVJ C01422 VJ=0.78
MOVL C01423 V=8.0
MOVJ C01424 VJ=0.78
MOVJ C01425 VJ=0.78
MOVJ C01426 VJ=0.78
MOVL C01427 V=8.0
MOVJ C01428 VJ=0.78
MOVJ C01429 VJ=0.78
MOVJ C01430 VJ=0.78
MOVL C01431 V=8.0
MOVJ C01432 VJ=0.78
MOVJ C01433 VJ=0.78
MOVJ C01434 VJ=0.78
MOVL C01435 V=8.0
MOVJ C01436 VJ=0.78
MOVJ C01437 VJ=0.78
MOVJ C01438 VJ=0.78
MOVL C01439 V=8.0
MOVJ C01440 VJ=0.78
MOVJ C01441 VJ=0.78
MOVJ C01442 VJ=0.78
MOVL C01443 V=8.0
MOVJ C01444 VJ=0.78
MOVJ C01445 VJ=0.78
MOVJ C01446 VJ=0.78
MOVL C01447 V=8.0
MOVJ C01448 VJ=0.78
MOVJ C01449 VJ=0.78
MOVJ C01450 VJ=0.78
MOVL C01451 V=8.0
MOVJ C01452 VJ=0.78
MOVJ C01453 VJ=0.78
MOVJ C01454 VJ=0.78
MOVL C01455 V=8.0
MOVJ C01456 VJ=0.78
MOVJ C01457 VJ=0.78
MOVJ C01458 VJ=0.78
MOVL C01459 V=8.0
MOVJ C01460 VJ=0.78
MOVJ C01461 VJ=0.78
MOVJ C01462 VJ=0.78
MOVL C01463 V=8.0
MOVJ C01464 VJ=0.78
MOVJ C01465 VJ=0.78
MOVJ C01466 VJ=0.78
MOVL C01467 V=8.0
MOVJ C01468 VJ=0.78
MOVJ C01469 VJ=0.78
MOVJ C01470 VJ=0.78
MOVL C01471 V=8.0
MOVJ C01472 VJ=0.78
MOVJ C01473 VJ=0.78
MOVJ C01474 VJ=0.78
MOVL C01475 V=8.0
MOVJ C01476 VJ=0.78
MOVJ C01477 VJ=0.78
MOVJ C01478 VJ=0.78
MOVL C01479 V=8.0
MOVJ C01480 VJ=0.78
MOVJ C01481 VJ=0.78
MOVJ C01482 VJ=0.78
MOVL C01483 V=8.0
MOVJ C01484 VJ=0.78
MOVJ C01485 VJ=0.78
MOVJ C01486 VJ=0.78
MOVL C01487 V=8.0
MOVJ C01488 VJ=0.78
MOVJ C01489 VJ=0.78
MOVJ C01490 VJ=0.78
MOVL C01491 V=8.0
MOVJ C01492 VJ=0.78
MOVJ C01493 VJ=0.78
MOVJ C01494 VJ=0.78
MOVL C01495 V=8.0
MOVJ C01496 VJ=0.78
MOVJ C01497 VJ=0.78
MOVJ C01498 VJ=0.78
MOVL C01499 V=8.0
MOVJ C01500 VJ=0.78
MOVJ C01501 VJ=0.78
MOVJ C01502 VJ=0.78
MOVL C01503 V=8.0
MOVJ C01504 VJ=0.78
MOVJ C01505 VJ=0.78
MOVJ C01506 VJ=0.78
MOVL C01507 V=8.0
MOVJ C01508 VJ=0.78
MOVJ C01509 VJ=0.78
MOVJ C01510 VJ=0.78
MOVL C01511 V=8.0
MOVJ C01512 VJ=0.78
MOVJ C01513 VJ=0.78
MOVJ C01514 VJ=0.78
MOVL C01515 V=8.0
MOVJ C01516 VJ=0.78
MOVJ C01517 VJ=0.78
MOVJ C01518 VJ=0.78
MOVL C01519 V=8.0
MOVJ C01520 VJ=0.78
MOVJ C01521 VJ=0.78
MOVJ C01522 VJ=0.78
MOVL C01523 V=8.0
MOVJ C01524 VJ=0.78
MOVJ C01525 VJ=0.78
MOVJ C01526 VJ=0.78
MOVL C01527 V=8.0
MOVJ C01528 VJ=0.78
MOVJ C01529 VJ=0.78
MOVJ C01530 VJ=0.78
MOVL C01531 V=8.0
MOVJ C01532 VJ=0.78
MOVJ C01533 VJ=0.78
MOVJ C01534 VJ=0.78
MOVL C01535 V=8.0
MOVJ C01536 VJ=0.78
MOVJ C01537 VJ=0.78
MOVJ C01538 VJ=0.78
MOVL C01539 V=8.0
MOVJ C01540 VJ=0.78
MOVJ C01541 VJ=0.78
MOVJ C01542 VJ=0.78
MOVL C01543 V=8.0
MOVJ C01544 VJ=0.78
MOVJ C01545 VJ=0.78
MOVJ C01546 VJ=0.78
MOVL C01547 V=8.0
MOVJ C01548 VJ=0.78
MOVJ C01549 VJ=0.78
MOVJ C01550 VJ=0.78
MOVL C01551 V=8.0
MOVJ C01552 VJ=0.78
MOVJ C01553 VJ=0.78
MOVJ C01554 VJ=0.78
MOVL C01555 V=8.0
MOVJ C01556 VJ=0.78
MOVJ C01557 VJ=0.78
MOVJ C01558 VJ=0.78
MOVL C01559 V=8.0
MOVJ C01560 VJ=0.78
MOVJ C01561 VJ=0.78
MOVJ C01562 VJ=0.78
MOVL C01563 V=8.0
MOVJ C01564 VJ=0.78
MOVJ C01565 VJ=0.78
MOVJ C01566 VJ=0.78
MOVL C01567 V=8.0
MOVJ C01568 VJ=0.78
MOVJ C01569 VJ=0.78
MOVJ C01570 VJ=0.78
MOVL C01571 V=8.0
MOVJ C01572 VJ=0.78
MOVJ C01573 VJ=0.78
MOVJ C01574 VJ=0.78
MOVL C01575 V=8.0
MOVJ C01576 VJ=0.78
MOVJ C01577 VJ=0.78
MOVJ C01578 VJ=0.78
MOVL C01579 V=8.0
MOVJ C01580 VJ=0.78
MOVJ C01581 VJ=0.78
MOVJ C01582 VJ=0.78
MOVL C01583 V=8.0
MOVJ C01584 VJ=0.78
MOVJ C01585 VJ=0.78
MOVJ C01586 VJ=0.78
MOVL C01587 V=8.0
MOVJ C01588 VJ=0.78
MOVJ C01589 VJ=0.78
MOVJ C01590 VJ=0.78
MOVL C01591 V=8.0
MOVJ C01592 VJ=0.78
MOVJ C01593 VJ=0.78
MOVJ C01594 VJ=0.78
MOVL C01595 V=8.0
MOVJ C01596 VJ=0.78
MOVJ C01597 VJ=0.78
MOVJ C01598 VJ=0.78
MOVL C01599 V=8.0
MOVJ C01600 VJ=0.78
MOVJ C01601 VJ=0.78
MOVJ C01602 VJ=0.78
MOVL C01603 V=8.0
MOVJ C01604 VJ=0.78
MOVJ C01605 VJ=0.78
MOVJ C01606 VJ=0.78
MOVL C01607 V=8.0
MOVJ C01608 VJ=0.78
MOVJ C01609 VJ=0.78
MOVJ C01610 VJ=0.78
MOVL C01611 V=8.0
MOVJ C01612 VJ=0.78
MOVJ C01613 VJ=0.78
MOVJ C01614 VJ=0.78
MOVL C01615 V=8.0
MOVJ C01616 VJ=0.78
MOVJ C01617 VJ=0.78
MOVJ C01618 VJ=0.78
MOVL C01619 V=8.0
MOVJ C01620 VJ=0.78
MOVJ C01621 VJ=0.78
MOVJ C01622 VJ=0.78
MOVL C01623 V=8.0
MOVJ C01624 VJ=0.78
MOVJ C01625 VJ=0.78
MOVJ C01626 VJ=0.78
MOVL C01627 V=8.0
MOVJ C01628 VJ=0.78
MOVJ C01629 VJ=0.78
MOVJ C01630 VJ=0.78
MOVL C01631 V=8.0
MOVJ C01632 VJ=0.78
MOVJ C01633 VJ=0.78
MOVJ C01634 VJ=0.78
MOVL C01635 V=8.0
MOVJ C01636 VJ=0.78
MOVJ C01637 VJ=0.78
MOVJ C01638 VJ=0.78
MOVL C01639 V=8.0
MOVJ C01640 VJ=0.78
MOVJ C01641 VJ=0.78
MOVJ C01642 VJ=0.78
MOVL C01643 V=8.0
MOVJ C01644 VJ=0.78
MOVJ C01645 VJ=0.78
MOVJ C01646 VJ=0.78
MOVL C01647 V=8.0
MOVJ C01648 VJ=0.78
MOVJ C01649 VJ=0.78
MOVJ C01650 VJ=0.78
MOVL C01651 V=8.0
MOVJ C01652 VJ=0.78
MOVJ C01653 VJ=0.78
MOVJ C01654 VJ=0.78
MOVL C01655 V=8.0
MOVJ C01656 VJ=0.78
MOVJ C01657 VJ=0.78
MOVJ C01658 VJ=0.78
MOVL C01659 V=8.0
MOVJ C01660 VJ=0.78
MOVJ C01661 VJ=0.78
MOVJ C01662 VJ=0.78
MOVL C01663 V=8.0
MOVJ C01664 VJ=0.78
MOVJ C01665 VJ=0.78
MOVJ C01666 VJ=0.78
MOVL C01667 V=8.0
MOVJ C01668 VJ=0.78
MOVJ C01669 VJ=0.78
MOVJ C01670 VJ=0.78
MOVL C01671 V=8.0
MOVJ C01672 VJ=0.78
MOVJ C01673 VJ=0.78
MOVJ C01674 VJ=0.78
MOVL C01675 V=8.0
MOVJ C01676 VJ=0.78
MOVJ C01677 VJ=0.78
MOVJ C01678 VJ=0.78
MOVL C01679 V=8.0
MOVJ C01680 VJ=0.78
MOVJ C01681 VJ=0.78
MOVJ C01682 VJ=0.78
MOVL C01683 V=8.0
MOVJ C01684 VJ=0.78
MOVJ C01685 VJ=0.78
MOVJ C01686 VJ=0.78
MOVL C01687 V=8.0
MOVJ C01688 VJ=0.78
MOVJ C01689 VJ=0.78
MOVJ C01690 VJ=0.78
MOVL C01691 V=8.0
MOVJ C01692 VJ=0.78
MOVJ C01693 VJ=0.78
MOVJ C01694 VJ=0.78
MOVL C01695 V=8.0
MOVJ C01696 VJ=0.78
MOVJ C01697 VJ=0.78
MOVJ C01698 VJ=0.78
MOVL C01699 V=8.0
MOVJ C01700 VJ=0.78
MOVJ C01701 VJ=0.78
MOVJ C01702 VJ=0.78
MOVL C01703 V=8.0
MOVJ C01704 VJ=0.78
MOVJ C01705 VJ=0.78
MOVJ C01706 VJ=0.78
MOVL C01707 V=8.0
MOVJ C01708 VJ=0.78
MOVJ C01709 VJ=0.78
MOVJ C01710 VJ=0.78
MOVL C01711 V=8.0
MOVJ C01712 VJ=0.78
MOVJ C01713 VJ=0.78
MOVJ C01714 VJ=0.78
MOVL C01715 V=8.0
MOVJ C01716 VJ=0.78
MOVJ C01717 VJ=0.78
MOVJ C01718 VJ=0.78
MOVL C01719 V=8.0
MOVJ C01720 VJ=0.78
MOVJ C01721 VJ=0.78
MOVJ C01722 VJ=0.78
MOVL C01723 V=8.0
MOVJ C01724 VJ=0.78
MOVJ C01725 VJ=0.78
MOVJ C01726 VJ=0.78
MOVL C01727 V=8.0
MOVJ C01728 VJ=0.78
MOVJ C01729 VJ=0.78
MOVJ C01730 VJ=0.78
MOVL C01731 V=8.0
MOVJ C01732 VJ=0.78
MOVJ C01733 VJ=0.78
MOVJ C01734 VJ=0.78
MOVL C01735 V=8.0
MOVJ C01736 VJ=0.78
MOVJ C01737 VJ=0.78
MOVJ C01738 VJ=0.78
MOVL C01739 V=8.0
MOVJ C01740 VJ=0.78
MOVJ C01741 VJ=0.78
MOVJ C01742 VJ=0.78
MOVL C01743 V=8.0
MOVJ C01744 VJ=0.78
MOVJ C01745 VJ=0.78
MOVJ C01746 VJ=0.78
MOVL C01747 V=8.0
MOVJ C01748 VJ=0.78
MOVJ C01749 VJ=0.78
MOVJ C01750 VJ=0.78
MOVL C01751 V=8.0
MOVJ C01752 VJ=0.78
MOVJ C01753 VJ=0.78
MOVJ C01754 VJ=0.78
MOVL C01755 V=8.0
MOVJ C01756 VJ=0.78
MOVJ C01757 VJ=0.78
MOVJ C01758 VJ=0.78
MOVL C01759 V=8.0
MOVJ C01760 VJ=0.78
MOVJ C01761 VJ=0.78
MOVJ C01762 VJ=0.78
MOVL C01763 V=8.0
MOVJ C01764 VJ=0.78
MOVJ C01765 VJ=0.78
MOVJ C01766 VJ=0.78
MOVL C01767 V=8.0
MOVJ C01768 VJ=0.78
MOVJ C01769 VJ=0.78
